// TIA Portal V20 export
FUNCTION "PMC_Map01" : Void   // FC5001, LAD
TITLE = GMPT Common Logic Template Version: G3.2
AUTHOR : JRose
FAMILY : CITI
NAME : MMG3.2
VERSION : 0.0
// stored: Namespace CITI_Logic, SetENOAutomatically false
   VAR_TEMP
      Team_Leader_Call : Bool;   // Unacknowledged Assistance Call is Active
      Flash_Red_Cmd : Bool;   // 1Hz Flasher
      Solid_Red_Cmd : Bool;   // 1Hz Flasher
      Flash_Yellow_Cmd : Bool;   // 1Hz Flasher
      Solid_Yellow_Cmd : Bool;   // 1Hz Flasher
      Flash_Green_Cmd : Bool;   // 1Hz Flasher
      Solid_Green_Cmd : Bool;   // 1Hz Flasher
      Flash_Blue_Cmd : Bool;   // 1Hz Flasher
      Solid_Blue_Cmd : Bool;   // 1Hz Flasher
      Flasher : Bool;   // 1Hz Flasher
      PUNData : String[18];
      FTQ_Reject_String : String[100];   // FTQ Data String PUN
      FTQ_Reject_Int : Int;   // FTQ Reject Integer
      LastPartTypeString : String[10];   // Last Part Type String
      EmptyPalletChar : Char;
      GM_PartNumber : String[8];
      OptionalData : String[9];
      HMI_Lite : Bool;
      HMI_Pro : Bool;
      TEMP_FOR_HMI_PRO : Bool;
      TEMP_FOR_UNIFIED_HMI : Bool;
      TEMP_HMI_INTERFACE : Bool;
      UNIFIED_HMI : Bool;
      OEM_ALARM_ID_from_ProDIAG : Int;
      Temp_Clock_Byte : Byte;
      TEMP_ALARM_FAULT : Array[0..499] of Word;
      Buffer_Count_Int : Int;
   END_VAR
   VAR_TEMP   // added for the SCL form of the ladder/FBD networks
      _w1 : Bool;
      _w2 : Bool;
      _w3 : Bool;
      _w4 : Bool;
      _w5 : Bool;
      _w6 : Bool;
      _w7 : Bool;
      _w8 : Bool;
      _w9 : Bool;
      _w10 : Bool;
      _w11 : Bool;
      _w12 : Bool;
   END_VAR
BEGIN

REGION Network 1
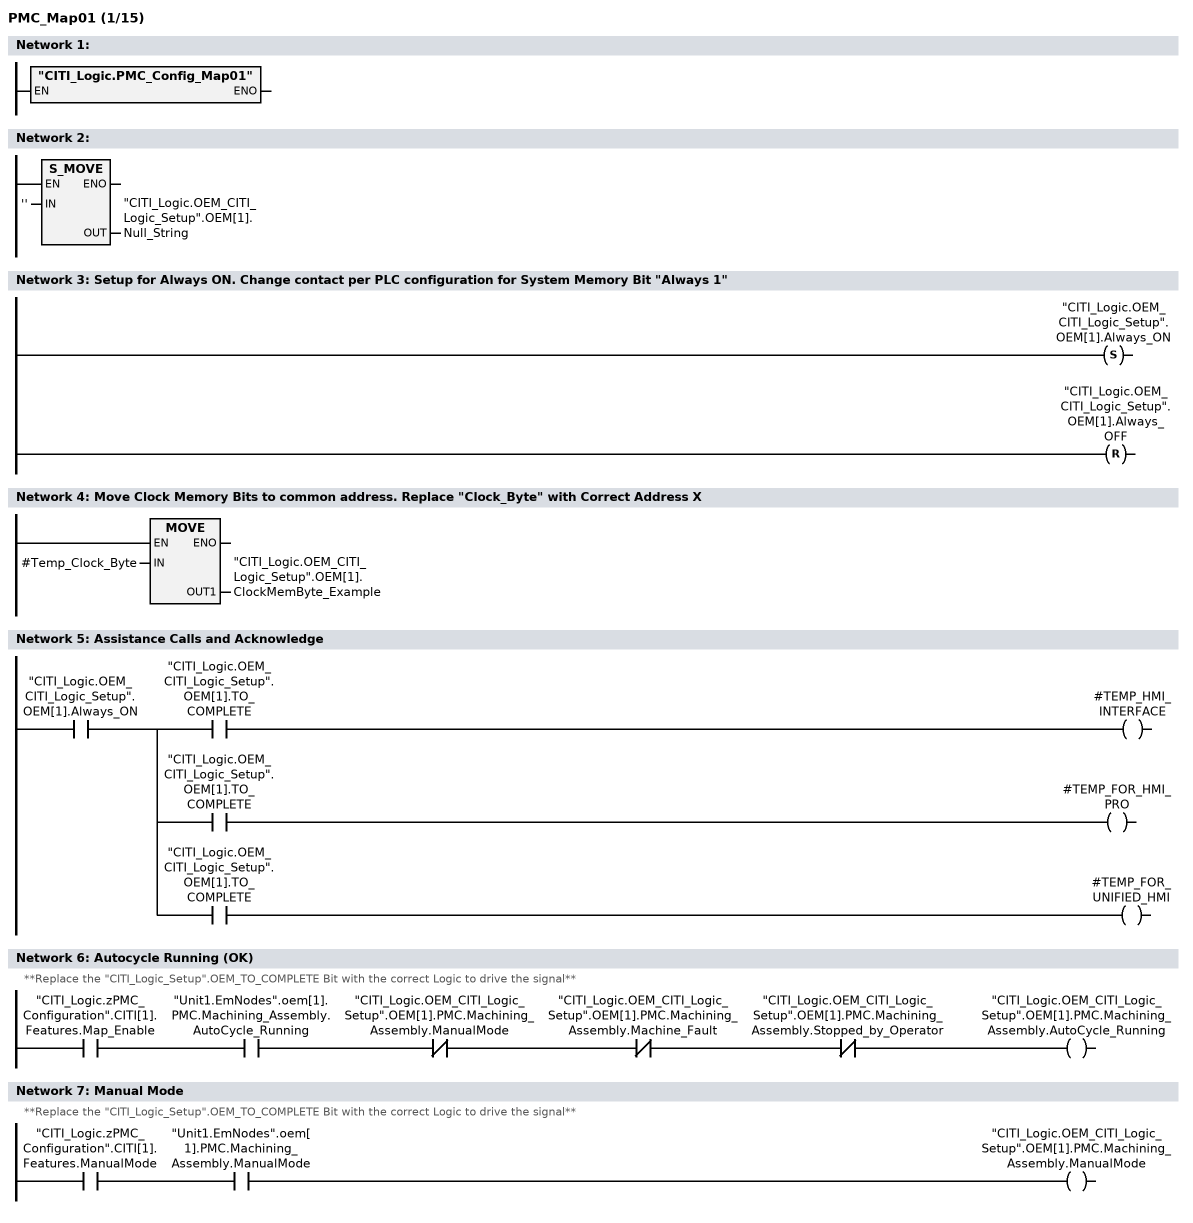
   RUNG wire#powerrail
      "CITI_Logic.PMC_Config_Map01"()
   END_RUNG
   // the same network as SCL:
   "CITI_Logic.PMC_Config_Map01"();
END_REGION

REGION Network 2
   RUNG wire#powerrail
      S_Move(in := '', out => "CITI_Logic.OEM_CITI_Logic_Setup".OEM[1].Null_String)
   END_RUNG
   // the same network as SCL:
   "CITI_Logic.OEM_CITI_Logic_Setup".OEM[1].Null_String := '';
END_REGION

REGION Network 3: Setup for Always ON. Change contact per PLC configuration for System Memory Bit "Always 1"
   RUNG wire#powerrail
      S_Coil( "CITI_Logic.OEM_CITI_Logic_Setup".OEM[1].Always_ON )
   END_RUNG
   RUNG wire#powerrail
      R_Coil( "CITI_Logic.OEM_CITI_Logic_Setup".OEM[1].Always_OFF )
   END_RUNG
   // the same network as SCL:
   "CITI_Logic.OEM_CITI_Logic_Setup".OEM[1].Always_ON := TRUE;
   "CITI_Logic.OEM_CITI_Logic_Setup".OEM[1].Always_OFF := FALSE;
END_REGION

REGION Network 4: Move Clock Memory Bits to common address. Replace "Clock_Byte" with Correct Address X
   RUNG wire#powerrail
      Move(in := #Temp_Clock_Byte, out1 => "CITI_Logic.OEM_CITI_Logic_Setup".OEM[1].ClockMemByte_Example)
   END_RUNG
   // the same network as SCL:
   "CITI_Logic.OEM_CITI_Logic_Setup".OEM[1].ClockMemByte_Example := #Temp_Clock_Byte;
END_REGION

REGION Network 5: Assistance Calls and Acknowledge
   RUNG wire#powerrail
      Contact( "CITI_Logic.OEM_CITI_Logic_Setup".OEM[1].Always_ON )
      wire#w1
      Contact( "CITI_Logic.OEM_CITI_Logic_Setup".OEM[1].TO_COMPLETE )
      Coil( #TEMP_HMI_INTERFACE )
   END_RUNG
   RUNG wire#w1
      Contact( "CITI_Logic.OEM_CITI_Logic_Setup".OEM[1].TO_COMPLETE )
      Coil( #TEMP_FOR_HMI_PRO )
   END_RUNG
   RUNG wire#w1
      Contact( "CITI_Logic.OEM_CITI_Logic_Setup".OEM[1].TO_COMPLETE )
      Coil( #TEMP_FOR_UNIFIED_HMI )
   END_RUNG
   // the same network as SCL:
   #TEMP_HMI_INTERFACE := "CITI_Logic.OEM_CITI_Logic_Setup".OEM[1].Always_ON AND "CITI_Logic.OEM_CITI_Logic_Setup".OEM[1].TO_COMPLETE;
   #TEMP_FOR_HMI_PRO := "CITI_Logic.OEM_CITI_Logic_Setup".OEM[1].Always_ON AND "CITI_Logic.OEM_CITI_Logic_Setup".OEM[1].TO_COMPLETE;
   #TEMP_FOR_UNIFIED_HMI := "CITI_Logic.OEM_CITI_Logic_Setup".OEM[1].Always_ON AND "CITI_Logic.OEM_CITI_Logic_Setup".OEM[1].TO_COMPLETE;
END_REGION

REGION Network 6: Autocycle Running (OK)
   // **Replace the "CITI_Logic_Setup".OEM_TO_COMPLETE Bit with the correct Logic to drive the signal**
   RUNG wire#powerrail
      Contact( "CITI_Logic.zPMC_Configuration".CITI[1].Features.Map_Enable )
      Contact( "Unit1.EmNodes".oem[1].PMC.Machining_Assembly.AutoCycle_Running )
      I_Contact( "CITI_Logic.OEM_CITI_Logic_Setup".OEM[1].PMC.Machining_Assembly.ManualMode )
      I_Contact( "CITI_Logic.OEM_CITI_Logic_Setup".OEM[1].PMC.Machining_Assembly.Machine_Fault )
      I_Contact( "CITI_Logic.OEM_CITI_Logic_Setup".OEM[1].PMC.Machining_Assembly.Stopped_by_Operator )
      Coil( "CITI_Logic.OEM_CITI_Logic_Setup".OEM[1].PMC.Machining_Assembly.AutoCycle_Running )
   END_RUNG
   // the same network as SCL:
   "CITI_Logic.OEM_CITI_Logic_Setup".OEM[1].PMC.Machining_Assembly.AutoCycle_Running := "CITI_Logic.zPMC_Configuration".CITI[1].Features.Map_Enable AND "Unit1.EmNodes".oem[1].PMC.Machining_Assembly.AutoCycle_Running AND NOT "CITI_Logic.OEM_CITI_Logic_Setup".OEM[1].PMC.Machining_Assembly.ManualMode AND NOT "CITI_Logic.OEM_CITI_Logic_Setup".OEM[1].PMC.Machining_Assembly.Machine_Fault AND NOT "CITI_Logic.OEM_CITI_Logic_Setup".OEM[1].PMC.Machining_Assembly.Stopped_by_Operator;
END_REGION

REGION Network 7: Manual Mode
   // **Replace the "CITI_Logic_Setup".OEM_TO_COMPLETE Bit with the correct Logic to drive the signal**
   RUNG wire#powerrail
      Contact( "CITI_Logic.zPMC_Configuration".CITI[1].Features.ManualMode )
      Contact( "Unit1.EmNodes".oem[1].PMC.Machining_Assembly.ManualMode )
      Coil( "CITI_Logic.OEM_CITI_Logic_Setup".OEM[1].PMC.Machining_Assembly.ManualMode )
   END_RUNG
   // the same network as SCL:
   "CITI_Logic.OEM_CITI_Logic_Setup".OEM[1].PMC.Machining_Assembly.ManualMode := "CITI_Logic.zPMC_Configuration".CITI[1].Features.ManualMode AND "Unit1.EmNodes".oem[1].PMC.Machining_Assembly.ManualMode;
END_REGION

REGION Network 8: Material Low (N/A)
   // **Replace the "CITI_Logic_Setup".OEM_TO_COMPLETE Bit with the correct Logic to drive the signal**
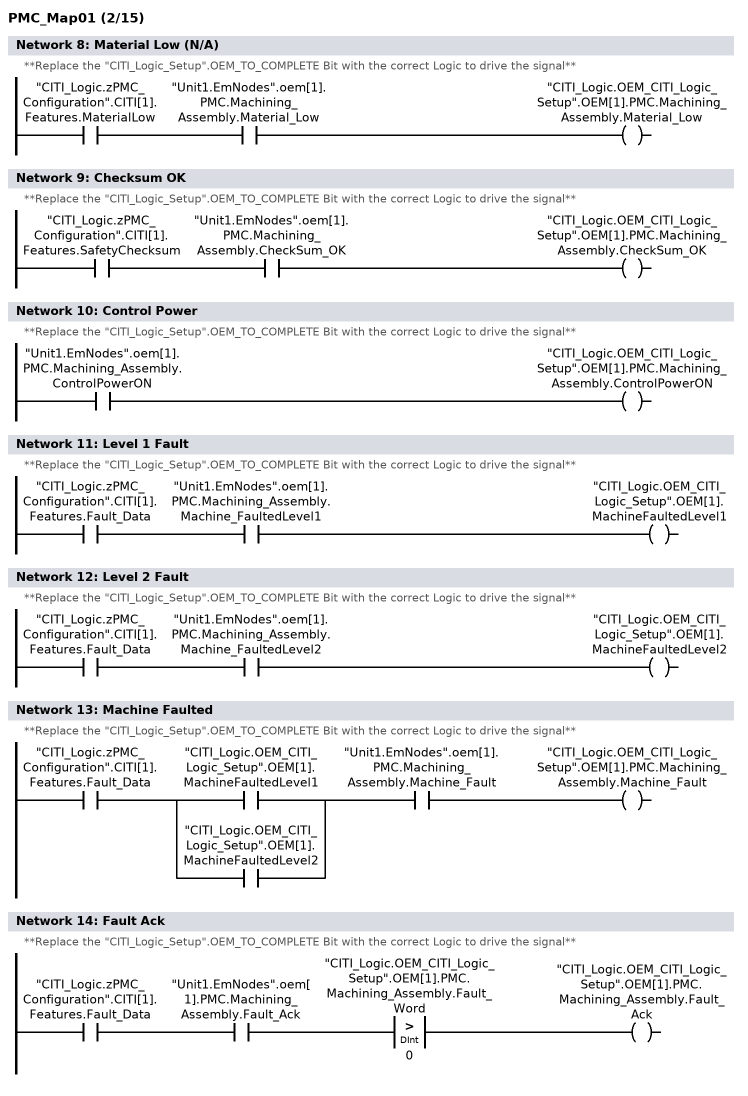
   RUNG wire#powerrail
      Contact( "CITI_Logic.zPMC_Configuration".CITI[1].Features.MaterialLow )
      Contact( "Unit1.EmNodes".oem[1].PMC.Machining_Assembly.Material_Low )
      Coil( "CITI_Logic.OEM_CITI_Logic_Setup".OEM[1].PMC.Machining_Assembly.Material_Low )
   END_RUNG
   // the same network as SCL:
   "CITI_Logic.OEM_CITI_Logic_Setup".OEM[1].PMC.Machining_Assembly.Material_Low := "CITI_Logic.zPMC_Configuration".CITI[1].Features.MaterialLow AND "Unit1.EmNodes".oem[1].PMC.Machining_Assembly.Material_Low;
END_REGION

REGION Network 9: Checksum OK
   // **Replace the "CITI_Logic_Setup".OEM_TO_COMPLETE Bit with the correct Logic to drive the signal**
   RUNG wire#powerrail
      Contact( "CITI_Logic.zPMC_Configuration".CITI[1].Features.SafetyChecksum )
      Contact( "Unit1.EmNodes".oem[1].PMC.Machining_Assembly.CheckSum_OK )
      Coil( "CITI_Logic.OEM_CITI_Logic_Setup".OEM[1].PMC.Machining_Assembly.CheckSum_OK )
   END_RUNG
   // the same network as SCL:
   "CITI_Logic.OEM_CITI_Logic_Setup".OEM[1].PMC.Machining_Assembly.CheckSum_OK := "CITI_Logic.zPMC_Configuration".CITI[1].Features.SafetyChecksum AND "Unit1.EmNodes".oem[1].PMC.Machining_Assembly.CheckSum_OK;
END_REGION

REGION Network 10: Control Power
   // **Replace the "CITI_Logic_Setup".OEM_TO_COMPLETE Bit with the correct Logic to drive the signal**
   RUNG wire#powerrail
      Contact( "Unit1.EmNodes".oem[1].PMC.Machining_Assembly.ControlPowerON )
      Coil( "CITI_Logic.OEM_CITI_Logic_Setup".OEM[1].PMC.Machining_Assembly.ControlPowerON )
   END_RUNG
   // the same network as SCL:
   "CITI_Logic.OEM_CITI_Logic_Setup".OEM[1].PMC.Machining_Assembly.ControlPowerON := "Unit1.EmNodes".oem[1].PMC.Machining_Assembly.ControlPowerON;
END_REGION

REGION Network 11: Level 1 Fault
   // **Replace the "CITI_Logic_Setup".OEM_TO_COMPLETE Bit with the correct Logic to drive the signal**
   RUNG wire#powerrail
      Contact( "CITI_Logic.zPMC_Configuration".CITI[1].Features.Fault_Data )
      Contact( "Unit1.EmNodes".oem[1].PMC.Machining_Assembly.Machine_FaultedLevel1 )
      Coil( "CITI_Logic.OEM_CITI_Logic_Setup".OEM[1].MachineFaultedLevel1 )
   END_RUNG
   // the same network as SCL:
   "CITI_Logic.OEM_CITI_Logic_Setup".OEM[1].MachineFaultedLevel1 := "CITI_Logic.zPMC_Configuration".CITI[1].Features.Fault_Data AND "Unit1.EmNodes".oem[1].PMC.Machining_Assembly.Machine_FaultedLevel1;
END_REGION

REGION Network 12: Level 2 Fault
   // **Replace the "CITI_Logic_Setup".OEM_TO_COMPLETE Bit with the correct Logic to drive the signal**
   RUNG wire#powerrail
      Contact( "CITI_Logic.zPMC_Configuration".CITI[1].Features.Fault_Data )
      Contact( "Unit1.EmNodes".oem[1].PMC.Machining_Assembly.Machine_FaultedLevel2 )
      Coil( "CITI_Logic.OEM_CITI_Logic_Setup".OEM[1].MachineFaultedLevel2 )
   END_RUNG
   // the same network as SCL:
   "CITI_Logic.OEM_CITI_Logic_Setup".OEM[1].MachineFaultedLevel2 := "CITI_Logic.zPMC_Configuration".CITI[1].Features.Fault_Data AND "Unit1.EmNodes".oem[1].PMC.Machining_Assembly.Machine_FaultedLevel2;
END_REGION

REGION Network 13: Machine Faulted
   // **Replace the "CITI_Logic_Setup".OEM_TO_COMPLETE Bit with the correct Logic to drive the signal**
   RUNG wire#powerrail
      Contact( "CITI_Logic.zPMC_Configuration".CITI[1].Features.Fault_Data )
      wire#w1
      Contact( "CITI_Logic.OEM_CITI_Logic_Setup".OEM[1].MachineFaultedLevel1 )
      wire#w2
      Contact( "Unit1.EmNodes".oem[1].PMC.Machining_Assembly.Machine_Fault )
      Coil( "CITI_Logic.OEM_CITI_Logic_Setup".OEM[1].PMC.Machining_Assembly.Machine_Fault )
   END_RUNG
   RUNG wire#w1
      Contact( "CITI_Logic.OEM_CITI_Logic_Setup".OEM[1].MachineFaultedLevel2 )
   END_RUNG wire#w2
   // the same network as SCL:
   "CITI_Logic.OEM_CITI_Logic_Setup".OEM[1].PMC.Machining_Assembly.Machine_Fault := "CITI_Logic.zPMC_Configuration".CITI[1].Features.Fault_Data AND ("CITI_Logic.OEM_CITI_Logic_Setup".OEM[1].MachineFaultedLevel1 OR "CITI_Logic.OEM_CITI_Logic_Setup".OEM[1].MachineFaultedLevel2) AND "Unit1.EmNodes".oem[1].PMC.Machining_Assembly.Machine_Fault;
END_REGION

REGION Network 14: Fault Ack
   // **Replace the "CITI_Logic_Setup".OEM_TO_COMPLETE Bit with the correct Logic to drive the signal**
   RUNG wire#powerrail
      Contact( "CITI_Logic.zPMC_Configuration".CITI[1].Features.Fault_Data )
      Contact( "Unit1.EmNodes".oem[1].PMC.Machining_Assembly.Fault_Ack )
      { S7_Templates := "SrcType := DInt" } GT_Contact(in1 := "CITI_Logic.OEM_CITI_Logic_Setup".OEM[1].PMC.Machining_Assembly.Fault_Word, in2 := 0)
      Coil( "CITI_Logic.OEM_CITI_Logic_Setup".OEM[1].PMC.Machining_Assembly.Fault_Ack )
   END_RUNG
   // the same network as SCL:
   "CITI_Logic.OEM_CITI_Logic_Setup".OEM[1].PMC.Machining_Assembly.Fault_Ack := "CITI_Logic.zPMC_Configuration".CITI[1].Features.Fault_Data AND "Unit1.EmNodes".oem[1].PMC.Machining_Assembly.Fault_Ack AND ("CITI_Logic.OEM_CITI_Logic_Setup".OEM[1].PMC.Machining_Assembly.Fault_Word > 0);
END_REGION

REGION Network 15: Stopped By Operator
   // **Replace the "CITI_Logic_Setup".OEM_TO_COMPLETE Bit with the correct Logic to drive the signal**
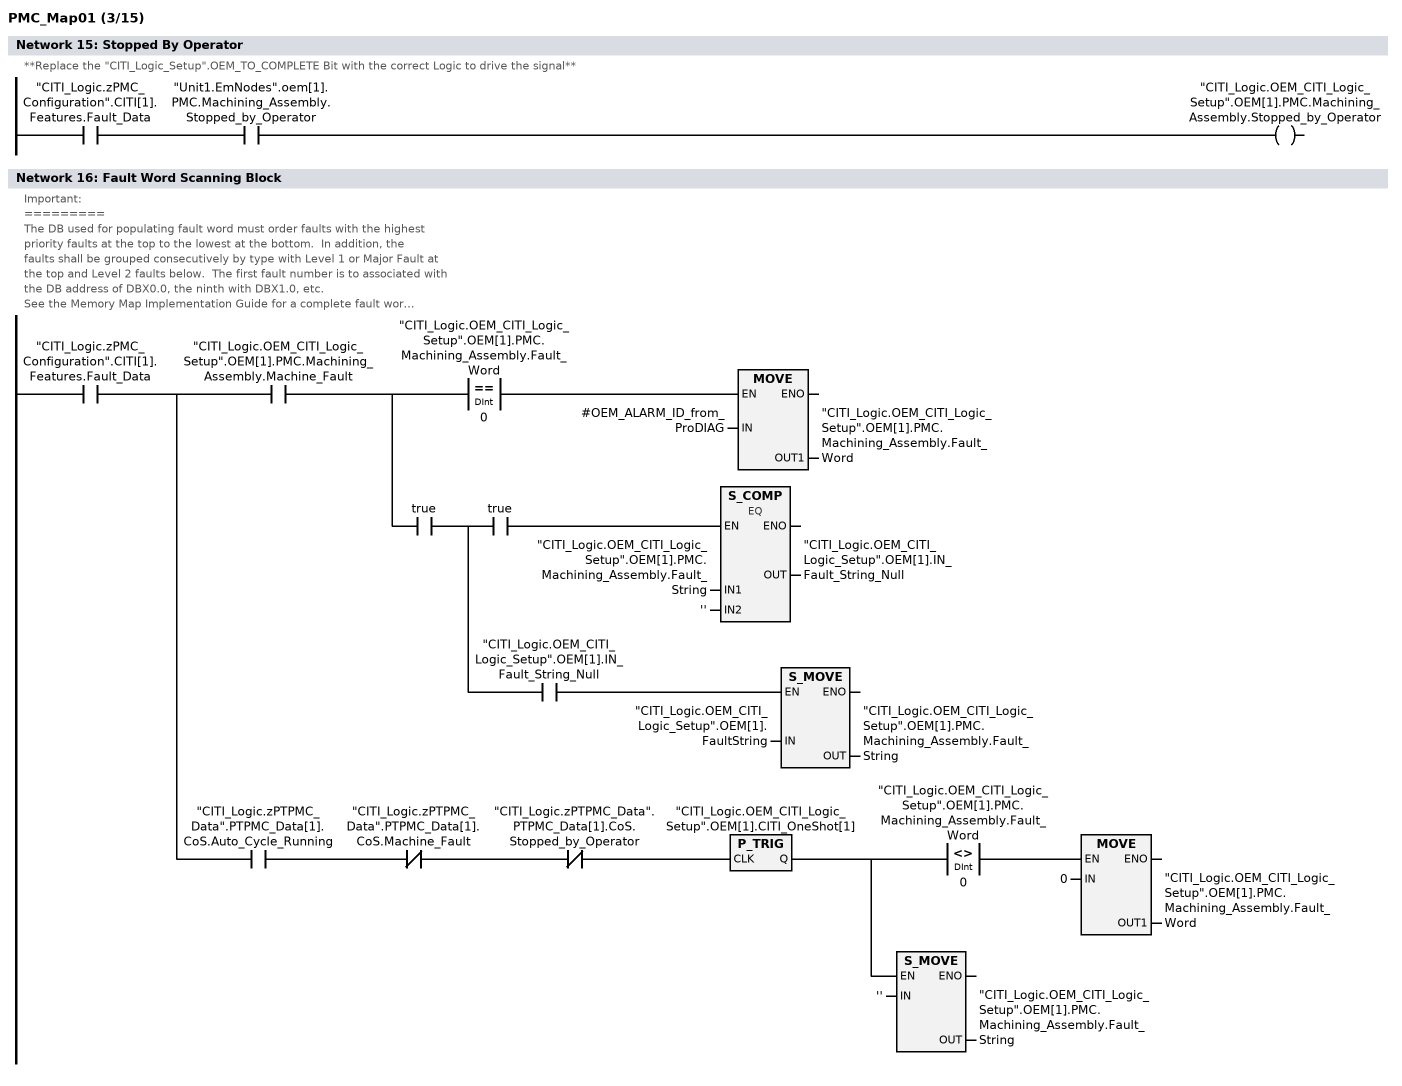
   RUNG wire#powerrail
      Contact( "CITI_Logic.zPMC_Configuration".CITI[1].Features.Fault_Data )
      Contact( "Unit1.EmNodes".oem[1].PMC.Machining_Assembly.Stopped_by_Operator )
      Coil( "CITI_Logic.OEM_CITI_Logic_Setup".OEM[1].PMC.Machining_Assembly.Stopped_by_Operator )
   END_RUNG
   // the same network as SCL:
   "CITI_Logic.OEM_CITI_Logic_Setup".OEM[1].PMC.Machining_Assembly.Stopped_by_Operator := "CITI_Logic.zPMC_Configuration".CITI[1].Features.Fault_Data AND "Unit1.EmNodes".oem[1].PMC.Machining_Assembly.Stopped_by_Operator;
END_REGION

REGION Network 16: Fault Word Scanning Block
   // Important:
   // =========
   // The DB used for populating fault word must order faults with the highest 
   // priority faults at the top to the lowest at the bottom.  In addition, the 
   // faults shall be grouped consecutively by type with Level 1 or Major Fault at 
   // the top and Level 2 faults below.  The first fault number is to associated with 
   // the DB address of DBX0.0, the ninth with DBX1.0, etc.
   // 
   // See the Memory Map Implementation Guide for a complete fault word 
   // implementation description and list of requirements.
   RUNG wire#powerrail
      Contact( "CITI_Logic.zPMC_Configuration".CITI[1].Features.Fault_Data )
      wire#w1
      Contact( "CITI_Logic.OEM_CITI_Logic_Setup".OEM[1].PMC.Machining_Assembly.Machine_Fault )
      wire#w2
      { S7_Templates := "SrcType := DInt" } EQ_Contact(in1 := "CITI_Logic.OEM_CITI_Logic_Setup".OEM[1].PMC.Machining_Assembly.Fault_Word, in2 := 0)
      Move(in := #OEM_ALARM_ID_from_ProDIAG, out1 => "CITI_Logic.OEM_CITI_Logic_Setup".OEM[1].PMC.Machining_Assembly.Fault_Word)
   END_RUNG
   RUNG wire#w2
      Contact( true )
      wire#w3
      Contact( true )
      { S7_Templates := "[relation := EQ, src_type := String]" } S_COMP(IN1 := "CITI_Logic.OEM_CITI_Logic_Setup".OEM[1].PMC.Machining_Assembly.Fault_String, IN2 := '', OUT => "CITI_Logic.OEM_CITI_Logic_Setup".OEM[1].IN_Fault_String_Null)
   END_RUNG
   RUNG wire#w3
      Contact( "CITI_Logic.OEM_CITI_Logic_Setup".OEM[1].IN_Fault_String_Null )
      S_Move(in := "CITI_Logic.OEM_CITI_Logic_Setup".OEM[1].FaultString, out => "CITI_Logic.OEM_CITI_Logic_Setup".OEM[1].PMC.Machining_Assembly.Fault_String)
   END_RUNG
   RUNG wire#w1
      Contact( "CITI_Logic.zPTPMC_Data".PTPMC_Data[1].CoS.Auto_Cycle_Running )
      I_Contact( "CITI_Logic.zPTPMC_Data".PTPMC_Data[1].CoS.Machine_Fault )
      I_Contact( "CITI_Logic.zPTPMC_Data".PTPMC_Data[1].CoS.Stopped_by_Operator )
      P_Trig( "CITI_Logic.OEM_CITI_Logic_Setup".OEM[1].CITI_OneShot[1] )
      wire#w4
      { S7_Templates := "SrcType := DInt" } NE_Contact(in1 := "CITI_Logic.OEM_CITI_Logic_Setup".OEM[1].PMC.Machining_Assembly.Fault_Word, in2 := 0)
      { S7_GenerateENO := "TRUE" } Move(in := 0, out1 => "CITI_Logic.OEM_CITI_Logic_Setup".OEM[1].PMC.Machining_Assembly.Fault_Word)
   END_RUNG
   RUNG wire#w4
      S_Move(in := '', out => "CITI_Logic.OEM_CITI_Logic_Setup".OEM[1].PMC.Machining_Assembly.Fault_String)
   END_RUNG
   // the same network as SCL:
   #_w1 := "CITI_Logic.zPMC_Configuration".CITI[1].Features.Fault_Data AND "CITI_Logic.OEM_CITI_Logic_Setup".OEM[1].PMC.Machining_Assembly.Machine_Fault;
   IF #_w1 AND ("CITI_Logic.OEM_CITI_Logic_Setup".OEM[1].PMC.Machining_Assembly.Fault_Word = 0) THEN
       "CITI_Logic.OEM_CITI_Logic_Setup".OEM[1].PMC.Machining_Assembly.Fault_Word := #OEM_ALARM_ID_from_ProDIAG;
   END_IF;
   #_w2 := #_w1 AND true;
   #_w3 := "CITI_Logic.zPMC_Configuration".CITI[1].Features.Fault_Data;
   IF #_w2 AND true THEN
       S_COMP(IN1 := "CITI_Logic.OEM_CITI_Logic_Setup".OEM[1].PMC.Machining_Assembly.Fault_String,
              IN2 := '',
              OUT => "CITI_Logic.OEM_CITI_Logic_Setup".OEM[1].IN_Fault_String_Null);
   END_IF;
   IF #_w2 AND "CITI_Logic.OEM_CITI_Logic_Setup".OEM[1].IN_Fault_String_Null THEN
       "CITI_Logic.OEM_CITI_Logic_Setup".OEM[1].PMC.Machining_Assembly.Fault_String := "CITI_Logic.OEM_CITI_Logic_Setup".OEM[1].FaultString;
   END_IF;
   #_w4 := #_w3 AND "CITI_Logic.zPTPMC_Data".PTPMC_Data[1].CoS.Auto_Cycle_Running AND NOT "CITI_Logic.zPTPMC_Data".PTPMC_Data[1].CoS.Machine_Fault AND NOT "CITI_Logic.zPTPMC_Data".PTPMC_Data[1].CoS.Stopped_by_Operator;
   #_w5 := #_w4 AND NOT "CITI_Logic.OEM_CITI_Logic_Setup".OEM[1].CITI_OneShot[1];   // rising edge
   "CITI_Logic.OEM_CITI_Logic_Setup".OEM[1].CITI_OneShot[1] := #_w4;
   IF #_w5 AND ("CITI_Logic.OEM_CITI_Logic_Setup".OEM[1].PMC.Machining_Assembly.Fault_Word <> 0) THEN
       "CITI_Logic.OEM_CITI_Logic_Setup".OEM[1].PMC.Machining_Assembly.Fault_Word := 0;
   END_IF;
   IF #_w5 THEN "CITI_Logic.OEM_CITI_Logic_Setup".OEM[1].PMC.Machining_Assembly.Fault_String := ''; END_IF;
END_REGION

REGION Network 17: Set up for Stopped by Other Map or Stopped with Unknown Fault
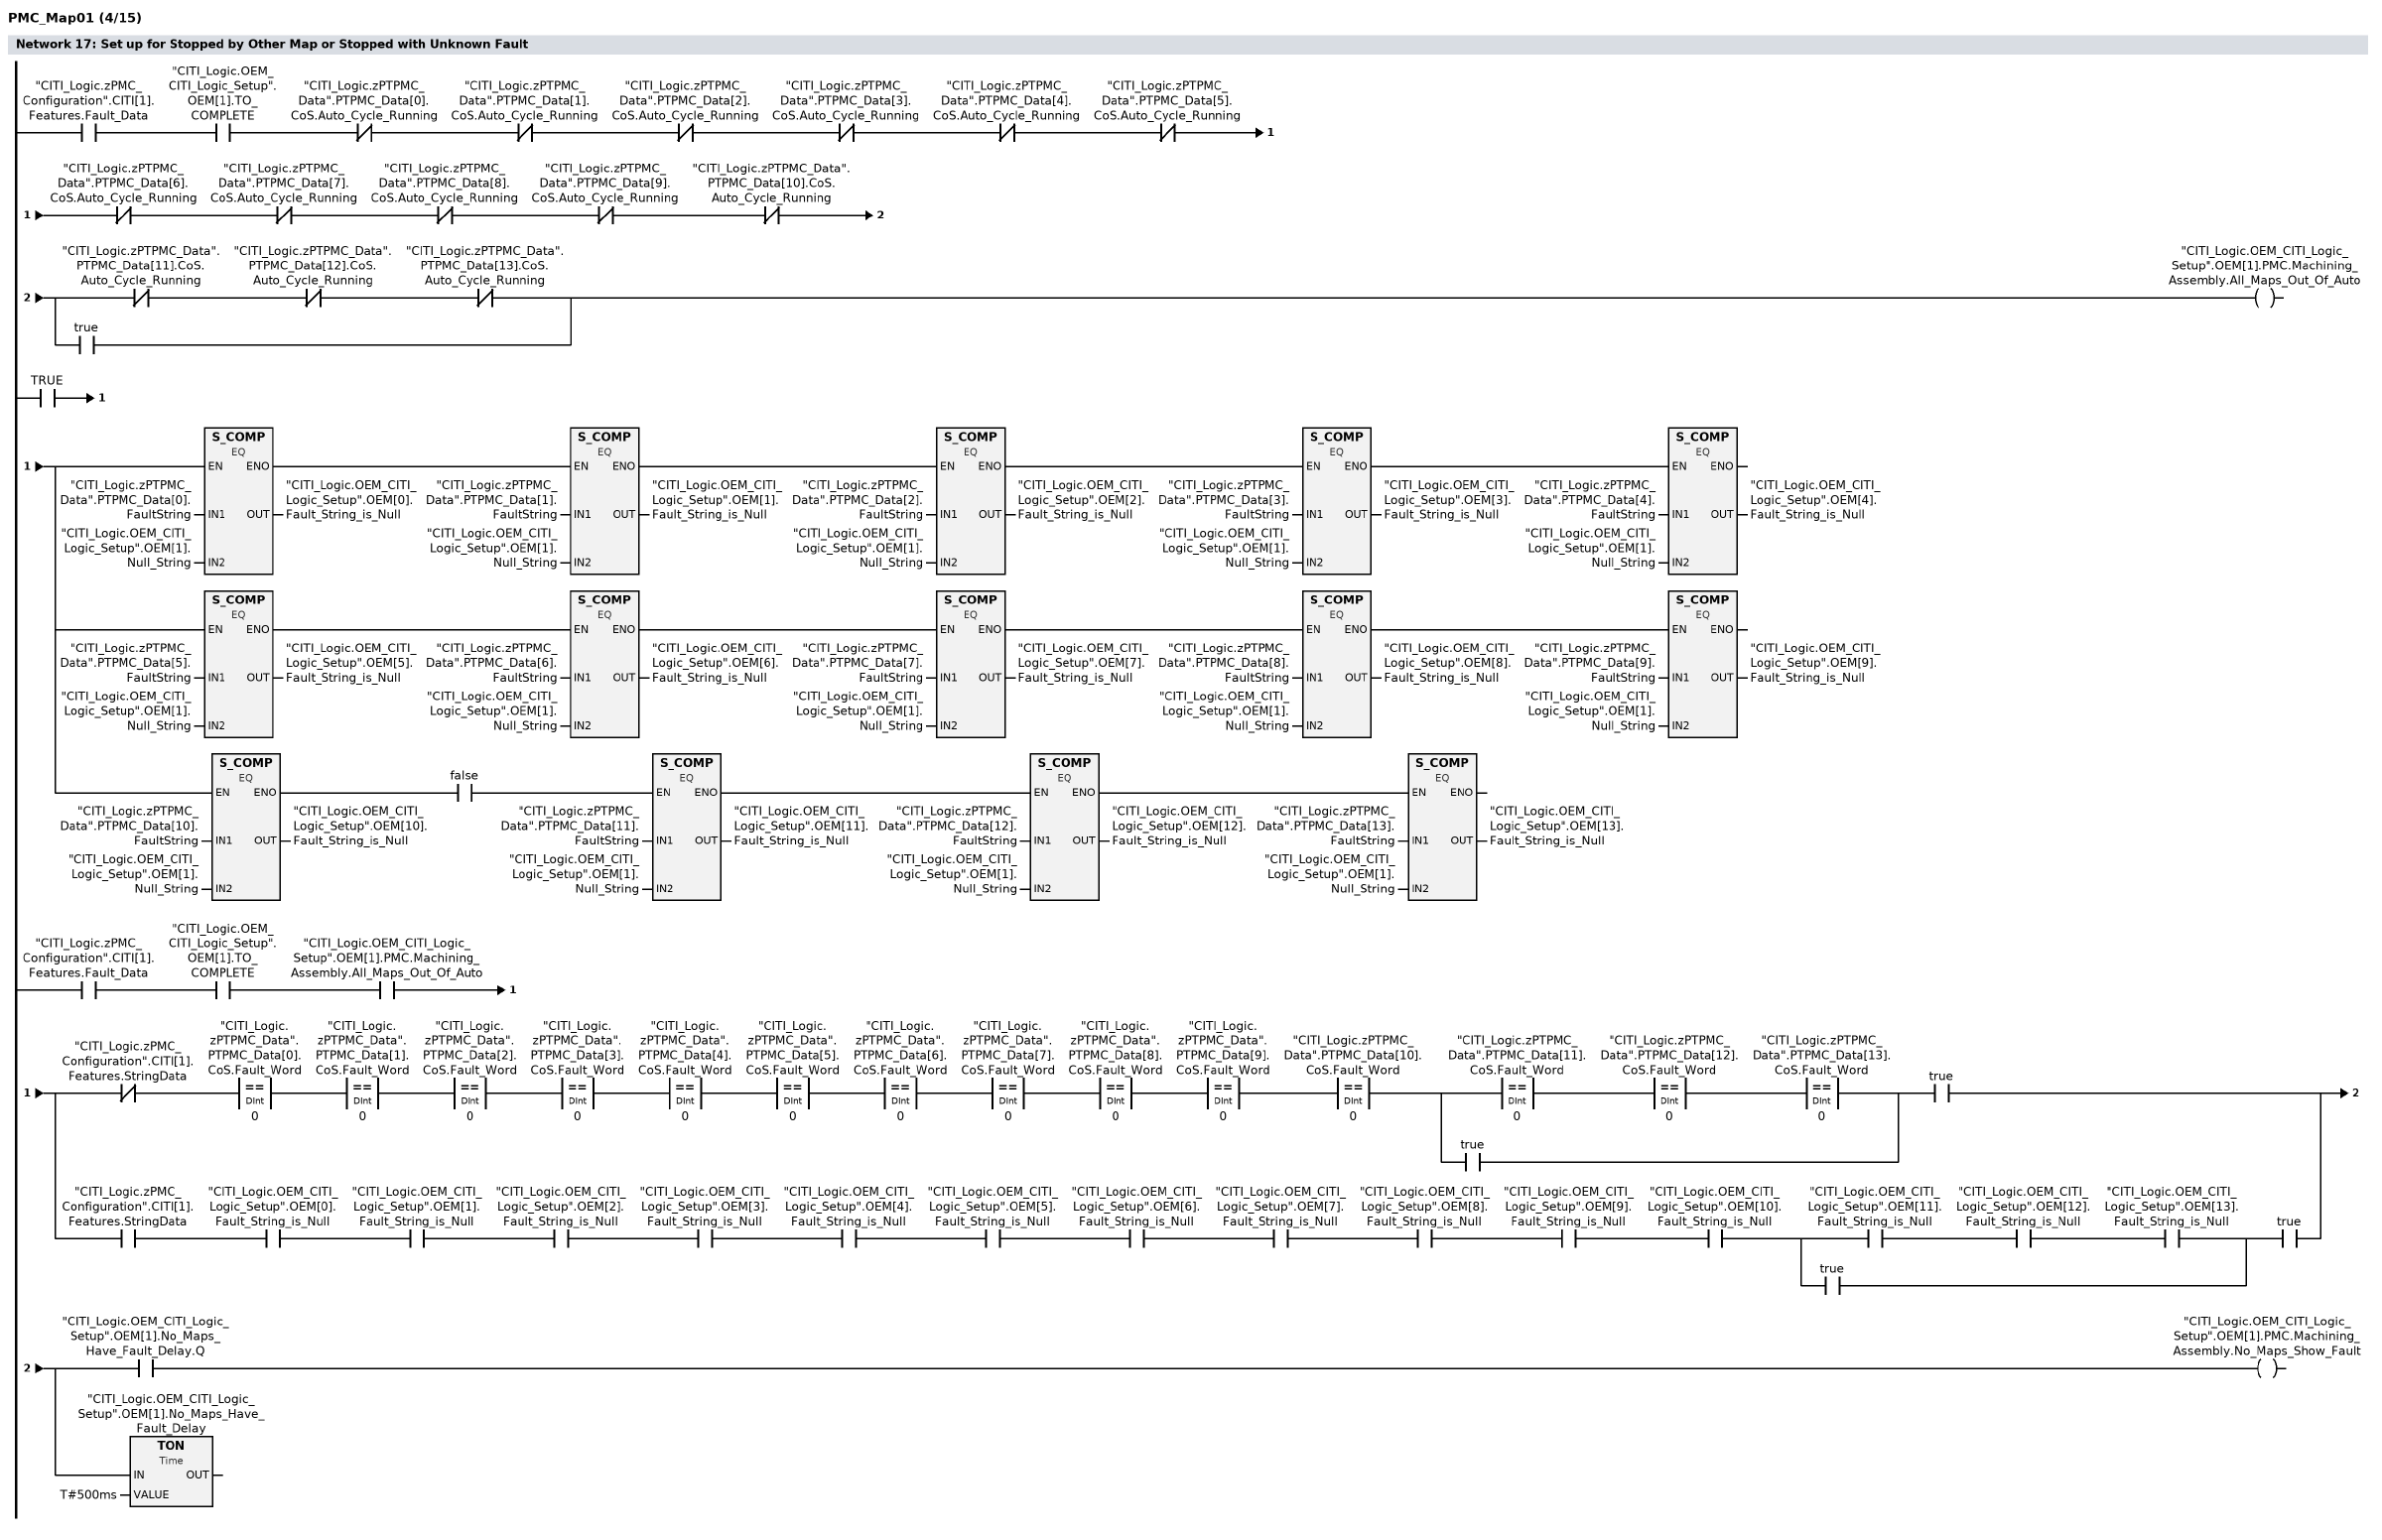
   "CITI_Logic.OEM_CITI_Logic_Setup".OEM[1].PMC.Machining_Assembly.All_Maps_Out_Of_Auto := "CITI_Logic.zPMC_Configuration".CITI[1].Features.Fault_Data AND "CITI_Logic.OEM_CITI_Logic_Setup".OEM[1].TO_COMPLETE AND NOT "CITI_Logic.zPTPMC_Data".PTPMC_Data[0].CoS.Auto_Cycle_Running AND NOT "CITI_Logic.zPTPMC_Data".PTPMC_Data[1].CoS.Auto_Cycle_Running AND NOT "CITI_Logic.zPTPMC_Data".PTPMC_Data[2].CoS.Auto_Cycle_Running AND NOT "CITI_Logic.zPTPMC_Data".PTPMC_Data[3].CoS.Auto_Cycle_Running AND NOT "CITI_Logic.zPTPMC_Data".PTPMC_Data[4].CoS.Auto_Cycle_Running AND NOT "CITI_Logic.zPTPMC_Data".PTPMC_Data[5].CoS.Auto_Cycle_Running AND NOT "CITI_Logic.zPTPMC_Data".PTPMC_Data[6].CoS.Auto_Cycle_Running AND NOT "CITI_Logic.zPTPMC_Data".PTPMC_Data[7].CoS.Auto_Cycle_Running AND NOT "CITI_Logic.zPTPMC_Data".PTPMC_Data[8].CoS.Auto_Cycle_Running AND NOT "CITI_Logic.zPTPMC_Data".PTPMC_Data[9].CoS.Auto_Cycle_Running AND NOT "CITI_Logic.zPTPMC_Data".PTPMC_Data[10].CoS.Auto_Cycle_Running AND ((NOT "CITI_Logic.zPTPMC_Data".PTPMC_Data[11].CoS.Auto_Cycle_Running AND NOT "CITI_Logic.zPTPMC_Data".PTPMC_Data[12].CoS.Auto_Cycle_Running AND NOT "CITI_Logic.zPTPMC_Data".PTPMC_Data[13].CoS.Auto_Cycle_Running) OR true);
   S_COMP(EN := TRUE,
          IN1 := "CITI_Logic.zPTPMC_Data".PTPMC_Data[0].FaultString,
          IN2 := "CITI_Logic.OEM_CITI_Logic_Setup".OEM[1].Null_String,
          OUT => "CITI_Logic.OEM_CITI_Logic_Setup".OEM[0].Fault_String_is_Null,
          ENO => #_w1);
   S_COMP(EN := #_w1,
          IN1 := "CITI_Logic.zPTPMC_Data".PTPMC_Data[1].FaultString,
          IN2 := "CITI_Logic.OEM_CITI_Logic_Setup".OEM[1].Null_String,
          OUT => "CITI_Logic.OEM_CITI_Logic_Setup".OEM[1].Fault_String_is_Null,
          ENO => #_w2);
   S_COMP(EN := #_w2,
          IN1 := "CITI_Logic.zPTPMC_Data".PTPMC_Data[2].FaultString,
          IN2 := "CITI_Logic.OEM_CITI_Logic_Setup".OEM[1].Null_String,
          OUT => "CITI_Logic.OEM_CITI_Logic_Setup".OEM[2].Fault_String_is_Null,
          ENO => #_w3);
   S_COMP(EN := #_w3,
          IN1 := "CITI_Logic.zPTPMC_Data".PTPMC_Data[3].FaultString,
          IN2 := "CITI_Logic.OEM_CITI_Logic_Setup".OEM[1].Null_String,
          OUT => "CITI_Logic.OEM_CITI_Logic_Setup".OEM[3].Fault_String_is_Null,
          ENO => #_w4);
   IF #_w4 THEN
       S_COMP(IN1 := "CITI_Logic.zPTPMC_Data".PTPMC_Data[4].FaultString,
              IN2 := "CITI_Logic.OEM_CITI_Logic_Setup".OEM[1].Null_String,
              OUT => "CITI_Logic.OEM_CITI_Logic_Setup".OEM[4].Fault_String_is_Null);
   END_IF;
   S_COMP(EN := TRUE,
          IN1 := "CITI_Logic.zPTPMC_Data".PTPMC_Data[5].FaultString,
          IN2 := "CITI_Logic.OEM_CITI_Logic_Setup".OEM[1].Null_String,
          OUT => "CITI_Logic.OEM_CITI_Logic_Setup".OEM[5].Fault_String_is_Null,
          ENO => #_w5);
   S_COMP(EN := #_w5,
          IN1 := "CITI_Logic.zPTPMC_Data".PTPMC_Data[6].FaultString,
          IN2 := "CITI_Logic.OEM_CITI_Logic_Setup".OEM[1].Null_String,
          OUT => "CITI_Logic.OEM_CITI_Logic_Setup".OEM[6].Fault_String_is_Null,
          ENO => #_w6);
   S_COMP(EN := #_w6,
          IN1 := "CITI_Logic.zPTPMC_Data".PTPMC_Data[7].FaultString,
          IN2 := "CITI_Logic.OEM_CITI_Logic_Setup".OEM[1].Null_String,
          OUT => "CITI_Logic.OEM_CITI_Logic_Setup".OEM[7].Fault_String_is_Null,
          ENO => #_w7);
   S_COMP(EN := #_w7,
          IN1 := "CITI_Logic.zPTPMC_Data".PTPMC_Data[8].FaultString,
          IN2 := "CITI_Logic.OEM_CITI_Logic_Setup".OEM[1].Null_String,
          OUT => "CITI_Logic.OEM_CITI_Logic_Setup".OEM[8].Fault_String_is_Null,
          ENO => #_w8);
   IF #_w8 THEN
       S_COMP(IN1 := "CITI_Logic.zPTPMC_Data".PTPMC_Data[9].FaultString,
              IN2 := "CITI_Logic.OEM_CITI_Logic_Setup".OEM[1].Null_String,
              OUT => "CITI_Logic.OEM_CITI_Logic_Setup".OEM[9].Fault_String_is_Null);
   END_IF;
   S_COMP(EN := TRUE,
          IN1 := "CITI_Logic.zPTPMC_Data".PTPMC_Data[10].FaultString,
          IN2 := "CITI_Logic.OEM_CITI_Logic_Setup".OEM[1].Null_String,
          OUT => "CITI_Logic.OEM_CITI_Logic_Setup".OEM[10].Fault_String_is_Null,
          ENO => #_w9);
   S_COMP(EN := #_w9 AND false,
          IN1 := "CITI_Logic.zPTPMC_Data".PTPMC_Data[11].FaultString,
          IN2 := "CITI_Logic.OEM_CITI_Logic_Setup".OEM[1].Null_String,
          OUT => "CITI_Logic.OEM_CITI_Logic_Setup".OEM[11].Fault_String_is_Null,
          ENO => #_w10);
   S_COMP(EN := #_w10,
          IN1 := "CITI_Logic.zPTPMC_Data".PTPMC_Data[12].FaultString,
          IN2 := "CITI_Logic.OEM_CITI_Logic_Setup".OEM[1].Null_String,
          OUT => "CITI_Logic.OEM_CITI_Logic_Setup".OEM[12].Fault_String_is_Null,
          ENO => #_w11);
   IF #_w11 THEN
       S_COMP(IN1 := "CITI_Logic.zPTPMC_Data".PTPMC_Data[13].FaultString,
              IN2 := "CITI_Logic.OEM_CITI_Logic_Setup".OEM[1].Null_String,
              OUT => "CITI_Logic.OEM_CITI_Logic_Setup".OEM[13].Fault_String_is_Null);
   END_IF;
   #_w12 := "CITI_Logic.zPMC_Configuration".CITI[1].Features.Fault_Data AND "CITI_Logic.OEM_CITI_Logic_Setup".OEM[1].TO_COMPLETE AND "CITI_Logic.OEM_CITI_Logic_Setup".OEM[1].PMC.Machining_Assembly.All_Maps_Out_Of_Auto AND ((NOT "CITI_Logic.zPMC_Configuration".CITI[1].Features.StringData AND ("CITI_Logic.zPTPMC_Data".PTPMC_Data[0].CoS.Fault_Word = 0) AND ("CITI_Logic.zPTPMC_Data".PTPMC_Data[1].CoS.Fault_Word = 0) AND ("CITI_Logic.zPTPMC_Data".PTPMC_Data[2].CoS.Fault_Word = 0) AND ("CITI_Logic.zPTPMC_Data".PTPMC_Data[3].CoS.Fault_Word = 0) AND ("CITI_Logic.zPTPMC_Data".PTPMC_Data[4].CoS.Fault_Word = 0) AND ("CITI_Logic.zPTPMC_Data".PTPMC_Data[5].CoS.Fault_Word = 0) AND ("CITI_Logic.zPTPMC_Data".PTPMC_Data[6].CoS.Fault_Word = 0) AND ("CITI_Logic.zPTPMC_Data".PTPMC_Data[7].CoS.Fault_Word = 0) AND ("CITI_Logic.zPTPMC_Data".PTPMC_Data[8].CoS.Fault_Word = 0) AND ("CITI_Logic.zPTPMC_Data".PTPMC_Data[9].CoS.Fault_Word = 0) AND ("CITI_Logic.zPTPMC_Data".PTPMC_Data[10].CoS.Fault_Word = 0) AND ((("CITI_Logic.zPTPMC_Data".PTPMC_Data[11].CoS.Fault_Word = 0) AND ("CITI_Logic.zPTPMC_Data".PTPMC_Data[12].CoS.Fault_Word = 0) AND ("CITI_Logic.zPTPMC_Data".PTPMC_Data[13].CoS.Fault_Word = 0)) OR true) AND true) OR ("CITI_Logic.zPMC_Configuration".CITI[1].Features.StringData AND "CITI_Logic.OEM_CITI_Logic_Setup".OEM[0].Fault_String_is_Null AND "CITI_Logic.OEM_CITI_Logic_Setup".OEM[1].Fault_String_is_Null AND "CITI_Logic.OEM_CITI_Logic_Setup".OEM[2].Fault_String_is_Null AND "CITI_Logic.OEM_CITI_Logic_Setup".OEM[3].Fault_String_is_Null AND "CITI_Logic.OEM_CITI_Logic_Setup".OEM[4].Fault_String_is_Null AND "CITI_Logic.OEM_CITI_Logic_Setup".OEM[5].Fault_String_is_Null AND "CITI_Logic.OEM_CITI_Logic_Setup".OEM[6].Fault_String_is_Null AND "CITI_Logic.OEM_CITI_Logic_Setup".OEM[7].Fault_String_is_Null AND "CITI_Logic.OEM_CITI_Logic_Setup".OEM[8].Fault_String_is_Null AND "CITI_Logic.OEM_CITI_Logic_Setup".OEM[9].Fault_String_is_Null AND "CITI_Logic.OEM_CITI_Logic_Setup".OEM[10].Fault_String_is_Null AND (("CITI_Logic.OEM_CITI_Logic_Setup".OEM[11].Fault_String_is_Null AND "CITI_Logic.OEM_CITI_Logic_Setup".OEM[12].Fault_String_is_Null AND "CITI_Logic.OEM_CITI_Logic_Setup".OEM[13].Fault_String_is_Null) OR true) AND true));
   "CITI_Logic.OEM_CITI_Logic_Setup".OEM[1].PMC.Machining_Assembly.No_Maps_Show_Fault := #_w12 AND "CITI_Logic.OEM_CITI_Logic_Setup".OEM[1].No_Maps_Have_Fault_Delay.Q;
   "CITI_Logic.OEM_CITI_Logic_Setup".OEM[1].No_Maps_Have_Fault_Delay.TON(IN := #_w12, PT := T#500ms);   // TON coil
END_REGION

REGION Network 18: Dry Cycle Mode
   // **Replace the "CITI_Logic_Setup".OEM_TO_COMPLETE Bit with the correct Logic to drive the signal**
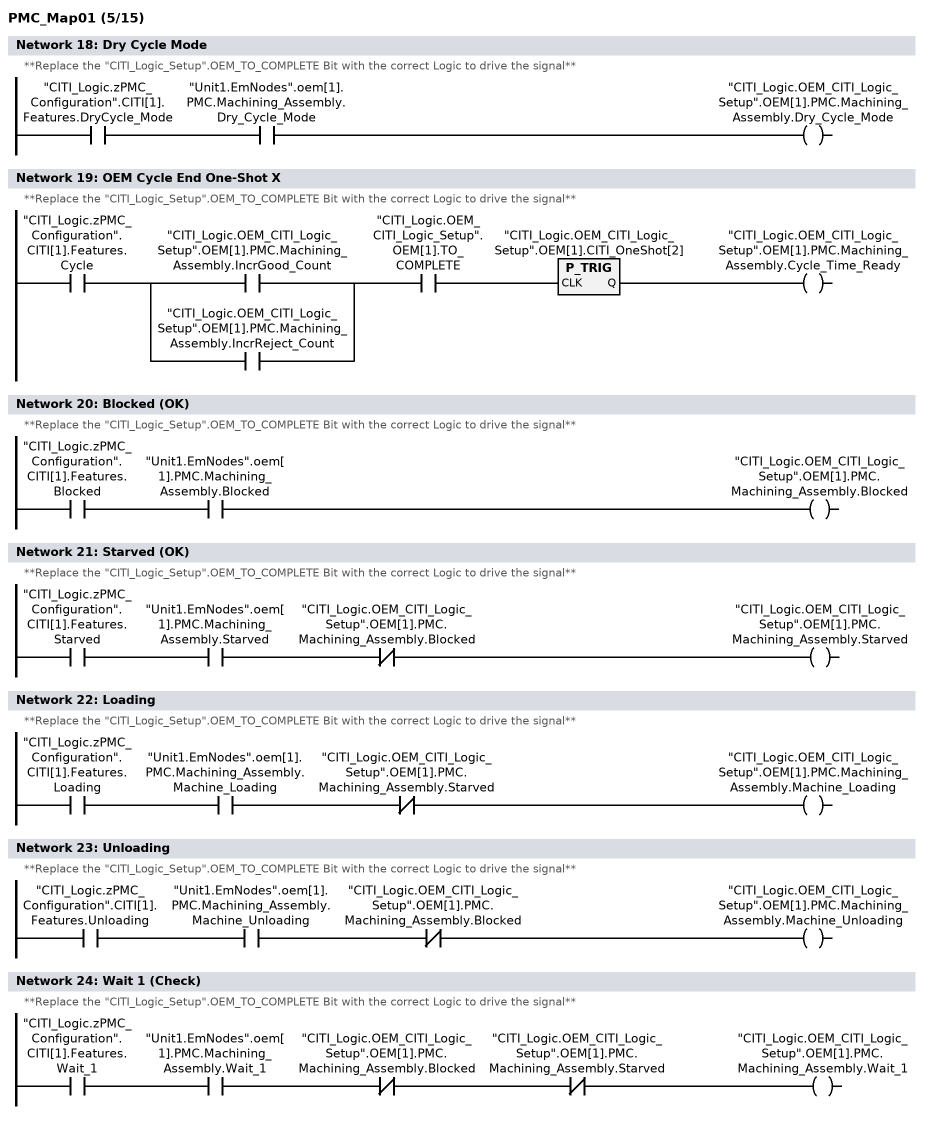
   RUNG wire#powerrail
      Contact( "CITI_Logic.zPMC_Configuration".CITI[1].Features.DryCycle_Mode )
      Contact( "Unit1.EmNodes".oem[1].PMC.Machining_Assembly.Dry_Cycle_Mode )
      Coil( "CITI_Logic.OEM_CITI_Logic_Setup".OEM[1].PMC.Machining_Assembly.Dry_Cycle_Mode )
   END_RUNG
   // the same network as SCL:
   "CITI_Logic.OEM_CITI_Logic_Setup".OEM[1].PMC.Machining_Assembly.Dry_Cycle_Mode := "CITI_Logic.zPMC_Configuration".CITI[1].Features.DryCycle_Mode AND "Unit1.EmNodes".oem[1].PMC.Machining_Assembly.Dry_Cycle_Mode;
END_REGION

REGION Network 19: OEM Cycle End One-Shot X
   // **Replace the "CITI_Logic_Setup".OEM_TO_COMPLETE Bit with the correct Logic to drive the signal**
   RUNG wire#powerrail
      Contact( "CITI_Logic.zPMC_Configuration".CITI[1].Features.Cycle )
      wire#w1
      Contact( "CITI_Logic.OEM_CITI_Logic_Setup".OEM[1].PMC.Machining_Assembly.IncrGood_Count )
      wire#w2
      Contact( "CITI_Logic.OEM_CITI_Logic_Setup".OEM[1].TO_COMPLETE )
      P_Trig( "CITI_Logic.OEM_CITI_Logic_Setup".OEM[1].CITI_OneShot[2] )
      Coil( "CITI_Logic.OEM_CITI_Logic_Setup".OEM[1].PMC.Machining_Assembly.Cycle_Time_Ready )
   END_RUNG
   RUNG wire#w1
      Contact( "CITI_Logic.OEM_CITI_Logic_Setup".OEM[1].PMC.Machining_Assembly.IncrReject_Count )
   END_RUNG wire#w2
   // the same network as SCL:
   #_w1 := "CITI_Logic.zPMC_Configuration".CITI[1].Features.Cycle AND ("CITI_Logic.OEM_CITI_Logic_Setup".OEM[1].PMC.Machining_Assembly.IncrGood_Count OR "CITI_Logic.OEM_CITI_Logic_Setup".OEM[1].PMC.Machining_Assembly.IncrReject_Count) AND "CITI_Logic.OEM_CITI_Logic_Setup".OEM[1].TO_COMPLETE;
   #_w2 := #_w1 AND NOT "CITI_Logic.OEM_CITI_Logic_Setup".OEM[1].CITI_OneShot[2];   // rising edge
   "CITI_Logic.OEM_CITI_Logic_Setup".OEM[1].CITI_OneShot[2] := #_w1;
   "CITI_Logic.OEM_CITI_Logic_Setup".OEM[1].PMC.Machining_Assembly.Cycle_Time_Ready := #_w2;
END_REGION

REGION Network 20: Blocked (OK)
   // **Replace the "CITI_Logic_Setup".OEM_TO_COMPLETE Bit with the correct Logic to drive the signal**
   RUNG wire#powerrail
      Contact( "CITI_Logic.zPMC_Configuration".CITI[1].Features.Blocked )
      Contact( "Unit1.EmNodes".oem[1].PMC.Machining_Assembly.Blocked )
      Coil( "CITI_Logic.OEM_CITI_Logic_Setup".OEM[1].PMC.Machining_Assembly.Blocked )
   END_RUNG
   // the same network as SCL:
   "CITI_Logic.OEM_CITI_Logic_Setup".OEM[1].PMC.Machining_Assembly.Blocked := "CITI_Logic.zPMC_Configuration".CITI[1].Features.Blocked AND "Unit1.EmNodes".oem[1].PMC.Machining_Assembly.Blocked;
END_REGION

REGION Network 21: Starved (OK)
   // **Replace the "CITI_Logic_Setup".OEM_TO_COMPLETE Bit with the correct Logic to drive the signal**
   RUNG wire#powerrail
      Contact( "CITI_Logic.zPMC_Configuration".CITI[1].Features.Starved )
      Contact( "Unit1.EmNodes".oem[1].PMC.Machining_Assembly.Starved )
      I_Contact( "CITI_Logic.OEM_CITI_Logic_Setup".OEM[1].PMC.Machining_Assembly.Blocked )
      Coil( "CITI_Logic.OEM_CITI_Logic_Setup".OEM[1].PMC.Machining_Assembly.Starved )
   END_RUNG
   // the same network as SCL:
   "CITI_Logic.OEM_CITI_Logic_Setup".OEM[1].PMC.Machining_Assembly.Starved := "CITI_Logic.zPMC_Configuration".CITI[1].Features.Starved AND "Unit1.EmNodes".oem[1].PMC.Machining_Assembly.Starved AND NOT "CITI_Logic.OEM_CITI_Logic_Setup".OEM[1].PMC.Machining_Assembly.Blocked;
END_REGION

REGION Network 22: Loading
   // **Replace the "CITI_Logic_Setup".OEM_TO_COMPLETE Bit with the correct Logic to drive the signal**
   RUNG wire#powerrail
      Contact( "CITI_Logic.zPMC_Configuration".CITI[1].Features.Loading )
      Contact( "Unit1.EmNodes".oem[1].PMC.Machining_Assembly.Machine_Loading )
      I_Contact( "CITI_Logic.OEM_CITI_Logic_Setup".OEM[1].PMC.Machining_Assembly.Starved )
      Coil( "CITI_Logic.OEM_CITI_Logic_Setup".OEM[1].PMC.Machining_Assembly.Machine_Loading )
   END_RUNG
   // the same network as SCL:
   "CITI_Logic.OEM_CITI_Logic_Setup".OEM[1].PMC.Machining_Assembly.Machine_Loading := "CITI_Logic.zPMC_Configuration".CITI[1].Features.Loading AND "Unit1.EmNodes".oem[1].PMC.Machining_Assembly.Machine_Loading AND NOT "CITI_Logic.OEM_CITI_Logic_Setup".OEM[1].PMC.Machining_Assembly.Starved;
END_REGION

REGION Network 23: Unloading
   // **Replace the "CITI_Logic_Setup".OEM_TO_COMPLETE Bit with the correct Logic to drive the signal**
   RUNG wire#powerrail
      Contact( "CITI_Logic.zPMC_Configuration".CITI[1].Features.Unloading )
      Contact( "Unit1.EmNodes".oem[1].PMC.Machining_Assembly.Machine_Unloading )
      I_Contact( "CITI_Logic.OEM_CITI_Logic_Setup".OEM[1].PMC.Machining_Assembly.Blocked )
      Coil( "CITI_Logic.OEM_CITI_Logic_Setup".OEM[1].PMC.Machining_Assembly.Machine_Unloading )
   END_RUNG
   // the same network as SCL:
   "CITI_Logic.OEM_CITI_Logic_Setup".OEM[1].PMC.Machining_Assembly.Machine_Unloading := "CITI_Logic.zPMC_Configuration".CITI[1].Features.Unloading AND "Unit1.EmNodes".oem[1].PMC.Machining_Assembly.Machine_Unloading AND NOT "CITI_Logic.OEM_CITI_Logic_Setup".OEM[1].PMC.Machining_Assembly.Blocked;
END_REGION

REGION Network 24: Wait 1 (Check)
   // **Replace the "CITI_Logic_Setup".OEM_TO_COMPLETE Bit with the correct Logic to drive the signal**
   RUNG wire#powerrail
      Contact( "CITI_Logic.zPMC_Configuration".CITI[1].Features.Wait_1 )
      Contact( "Unit1.EmNodes".oem[1].PMC.Machining_Assembly.Wait_1 )
      I_Contact( "CITI_Logic.OEM_CITI_Logic_Setup".OEM[1].PMC.Machining_Assembly.Blocked )
      I_Contact( "CITI_Logic.OEM_CITI_Logic_Setup".OEM[1].PMC.Machining_Assembly.Starved )
      Coil( "CITI_Logic.OEM_CITI_Logic_Setup".OEM[1].PMC.Machining_Assembly.Wait_1 )
   END_RUNG
   // the same network as SCL:
   "CITI_Logic.OEM_CITI_Logic_Setup".OEM[1].PMC.Machining_Assembly.Wait_1 := "CITI_Logic.zPMC_Configuration".CITI[1].Features.Wait_1 AND "Unit1.EmNodes".oem[1].PMC.Machining_Assembly.Wait_1 AND NOT "CITI_Logic.OEM_CITI_Logic_Setup".OEM[1].PMC.Machining_Assembly.Blocked AND NOT "CITI_Logic.OEM_CITI_Logic_Setup".OEM[1].PMC.Machining_Assembly.Starved;
END_REGION

REGION Network 25: Wait 2 (Check)
   // **Replace the "CITI_Logic_Setup".OEM_TO_COMPLETE Bit with the correct Logic to drive the signal**
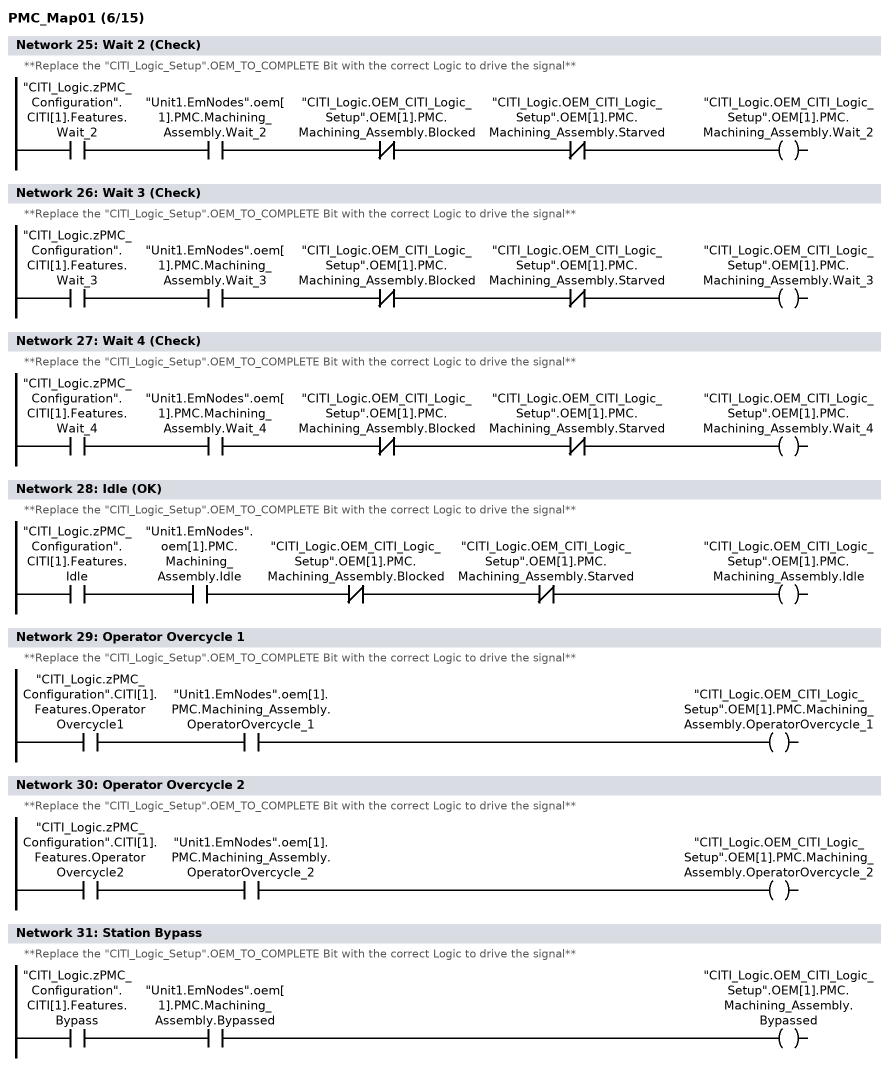
   RUNG wire#powerrail
      Contact( "CITI_Logic.zPMC_Configuration".CITI[1].Features.Wait_2 )
      Contact( "Unit1.EmNodes".oem[1].PMC.Machining_Assembly.Wait_2 )
      I_Contact( "CITI_Logic.OEM_CITI_Logic_Setup".OEM[1].PMC.Machining_Assembly.Blocked )
      I_Contact( "CITI_Logic.OEM_CITI_Logic_Setup".OEM[1].PMC.Machining_Assembly.Starved )
      Coil( "CITI_Logic.OEM_CITI_Logic_Setup".OEM[1].PMC.Machining_Assembly.Wait_2 )
   END_RUNG
   // the same network as SCL:
   "CITI_Logic.OEM_CITI_Logic_Setup".OEM[1].PMC.Machining_Assembly.Wait_2 := "CITI_Logic.zPMC_Configuration".CITI[1].Features.Wait_2 AND "Unit1.EmNodes".oem[1].PMC.Machining_Assembly.Wait_2 AND NOT "CITI_Logic.OEM_CITI_Logic_Setup".OEM[1].PMC.Machining_Assembly.Blocked AND NOT "CITI_Logic.OEM_CITI_Logic_Setup".OEM[1].PMC.Machining_Assembly.Starved;
END_REGION

REGION Network 26: Wait 3 (Check)
   // **Replace the "CITI_Logic_Setup".OEM_TO_COMPLETE Bit with the correct Logic to drive the signal**
   RUNG wire#powerrail
      Contact( "CITI_Logic.zPMC_Configuration".CITI[1].Features.Wait_3 )
      Contact( "Unit1.EmNodes".oem[1].PMC.Machining_Assembly.Wait_3 )
      I_Contact( "CITI_Logic.OEM_CITI_Logic_Setup".OEM[1].PMC.Machining_Assembly.Blocked )
      I_Contact( "CITI_Logic.OEM_CITI_Logic_Setup".OEM[1].PMC.Machining_Assembly.Starved )
      Coil( "CITI_Logic.OEM_CITI_Logic_Setup".OEM[1].PMC.Machining_Assembly.Wait_3 )
   END_RUNG
   // the same network as SCL:
   "CITI_Logic.OEM_CITI_Logic_Setup".OEM[1].PMC.Machining_Assembly.Wait_3 := "CITI_Logic.zPMC_Configuration".CITI[1].Features.Wait_3 AND "Unit1.EmNodes".oem[1].PMC.Machining_Assembly.Wait_3 AND NOT "CITI_Logic.OEM_CITI_Logic_Setup".OEM[1].PMC.Machining_Assembly.Blocked AND NOT "CITI_Logic.OEM_CITI_Logic_Setup".OEM[1].PMC.Machining_Assembly.Starved;
END_REGION

REGION Network 27: Wait 4 (Check)
   // **Replace the "CITI_Logic_Setup".OEM_TO_COMPLETE Bit with the correct Logic to drive the signal**
   RUNG wire#powerrail
      Contact( "CITI_Logic.zPMC_Configuration".CITI[1].Features.Wait_4 )
      Contact( "Unit1.EmNodes".oem[1].PMC.Machining_Assembly.Wait_4 )
      I_Contact( "CITI_Logic.OEM_CITI_Logic_Setup".OEM[1].PMC.Machining_Assembly.Blocked )
      I_Contact( "CITI_Logic.OEM_CITI_Logic_Setup".OEM[1].PMC.Machining_Assembly.Starved )
      Coil( "CITI_Logic.OEM_CITI_Logic_Setup".OEM[1].PMC.Machining_Assembly.Wait_4 )
   END_RUNG
   // the same network as SCL:
   "CITI_Logic.OEM_CITI_Logic_Setup".OEM[1].PMC.Machining_Assembly.Wait_4 := "CITI_Logic.zPMC_Configuration".CITI[1].Features.Wait_4 AND "Unit1.EmNodes".oem[1].PMC.Machining_Assembly.Wait_4 AND NOT "CITI_Logic.OEM_CITI_Logic_Setup".OEM[1].PMC.Machining_Assembly.Blocked AND NOT "CITI_Logic.OEM_CITI_Logic_Setup".OEM[1].PMC.Machining_Assembly.Starved;
END_REGION

REGION Network 28: Idle (OK)
   // **Replace the "CITI_Logic_Setup".OEM_TO_COMPLETE Bit with the correct Logic to drive the signal**
   RUNG wire#powerrail
      Contact( "CITI_Logic.zPMC_Configuration".CITI[1].Features.Idle )
      Contact( "Unit1.EmNodes".oem[1].PMC.Machining_Assembly.Idle )
      I_Contact( "CITI_Logic.OEM_CITI_Logic_Setup".OEM[1].PMC.Machining_Assembly.Blocked )
      I_Contact( "CITI_Logic.OEM_CITI_Logic_Setup".OEM[1].PMC.Machining_Assembly.Starved )
      Coil( "CITI_Logic.OEM_CITI_Logic_Setup".OEM[1].PMC.Machining_Assembly.Idle )
   END_RUNG
   // the same network as SCL:
   "CITI_Logic.OEM_CITI_Logic_Setup".OEM[1].PMC.Machining_Assembly.Idle := "CITI_Logic.zPMC_Configuration".CITI[1].Features.Idle AND "Unit1.EmNodes".oem[1].PMC.Machining_Assembly.Idle AND NOT "CITI_Logic.OEM_CITI_Logic_Setup".OEM[1].PMC.Machining_Assembly.Blocked AND NOT "CITI_Logic.OEM_CITI_Logic_Setup".OEM[1].PMC.Machining_Assembly.Starved;
END_REGION

REGION Network 29: Operator Overcycle 1
   // **Replace the "CITI_Logic_Setup".OEM_TO_COMPLETE Bit with the correct Logic to drive the signal**
   RUNG wire#powerrail
      Contact( "CITI_Logic.zPMC_Configuration".CITI[1].Features.OperatorOvercycle1 )
      Contact( "Unit1.EmNodes".oem[1].PMC.Machining_Assembly.OperatorOvercycle_1 )
      Coil( "CITI_Logic.OEM_CITI_Logic_Setup".OEM[1].PMC.Machining_Assembly.OperatorOvercycle_1 )
   END_RUNG
   // the same network as SCL:
   "CITI_Logic.OEM_CITI_Logic_Setup".OEM[1].PMC.Machining_Assembly.OperatorOvercycle_1 := "CITI_Logic.zPMC_Configuration".CITI[1].Features.OperatorOvercycle1 AND "Unit1.EmNodes".oem[1].PMC.Machining_Assembly.OperatorOvercycle_1;
END_REGION

REGION Network 30: Operator Overcycle 2
   // **Replace the "CITI_Logic_Setup".OEM_TO_COMPLETE Bit with the correct Logic to drive the signal**
   RUNG wire#powerrail
      Contact( "CITI_Logic.zPMC_Configuration".CITI[1].Features.OperatorOvercycle2 )
      Contact( "Unit1.EmNodes".oem[1].PMC.Machining_Assembly.OperatorOvercycle_2 )
      Coil( "CITI_Logic.OEM_CITI_Logic_Setup".OEM[1].PMC.Machining_Assembly.OperatorOvercycle_2 )
   END_RUNG
   // the same network as SCL:
   "CITI_Logic.OEM_CITI_Logic_Setup".OEM[1].PMC.Machining_Assembly.OperatorOvercycle_2 := "CITI_Logic.zPMC_Configuration".CITI[1].Features.OperatorOvercycle2 AND "Unit1.EmNodes".oem[1].PMC.Machining_Assembly.OperatorOvercycle_2;
END_REGION

REGION Network 31: Station Bypass
   // **Replace the "CITI_Logic_Setup".OEM_TO_COMPLETE Bit with the correct Logic to drive the signal**
   RUNG wire#powerrail
      Contact( "CITI_Logic.zPMC_Configuration".CITI[1].Features.Bypass )
      Contact( "Unit1.EmNodes".oem[1].PMC.Machining_Assembly.Bypassed )
      Coil( "CITI_Logic.OEM_CITI_Logic_Setup".OEM[1].PMC.Machining_Assembly.Bypassed )
   END_RUNG
   // the same network as SCL:
   "CITI_Logic.OEM_CITI_Logic_Setup".OEM[1].PMC.Machining_Assembly.Bypassed := "CITI_Logic.zPMC_Configuration".CITI[1].Features.Bypass AND "Unit1.EmNodes".oem[1].PMC.Machining_Assembly.Bypassed;
END_REGION

REGION Network 32: Good Count Trigger
   // **Replace the "CITI_Logic_Setup".OEM_TO_COMPLETE Bit with the correct Logic to drive the signal**
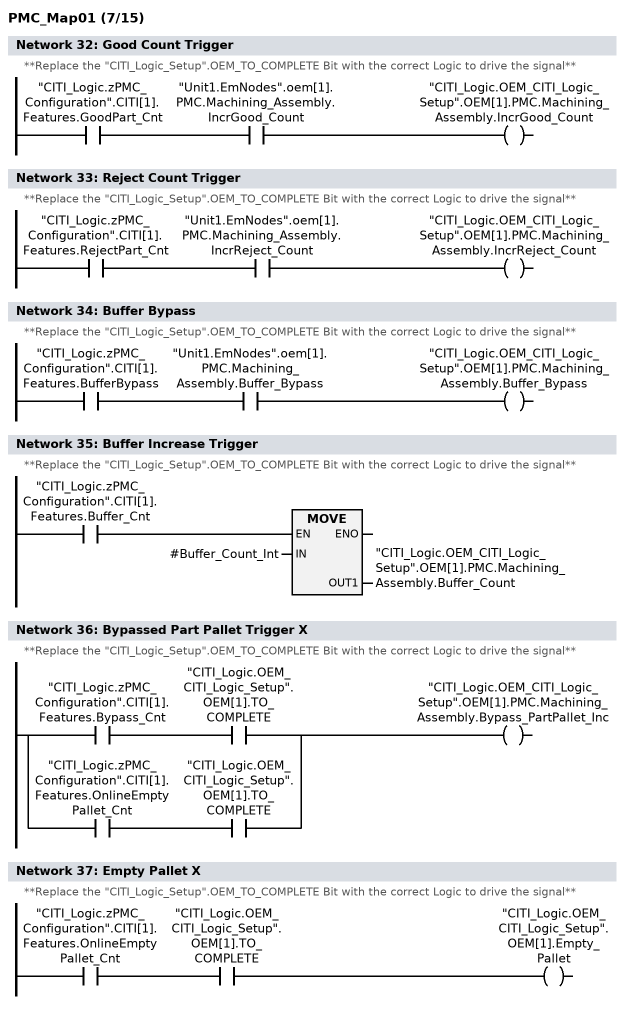
   RUNG wire#powerrail
      Contact( "CITI_Logic.zPMC_Configuration".CITI[1].Features.GoodPart_Cnt )
      Contact( "Unit1.EmNodes".oem[1].PMC.Machining_Assembly.IncrGood_Count )
      Coil( "CITI_Logic.OEM_CITI_Logic_Setup".OEM[1].PMC.Machining_Assembly.IncrGood_Count )
   END_RUNG
   // the same network as SCL:
   "CITI_Logic.OEM_CITI_Logic_Setup".OEM[1].PMC.Machining_Assembly.IncrGood_Count := "CITI_Logic.zPMC_Configuration".CITI[1].Features.GoodPart_Cnt AND "Unit1.EmNodes".oem[1].PMC.Machining_Assembly.IncrGood_Count;
END_REGION

REGION Network 33: Reject Count Trigger
   // **Replace the "CITI_Logic_Setup".OEM_TO_COMPLETE Bit with the correct Logic to drive the signal**
   RUNG wire#powerrail
      Contact( "CITI_Logic.zPMC_Configuration".CITI[1].Features.RejectPart_Cnt )
      Contact( "Unit1.EmNodes".oem[1].PMC.Machining_Assembly.IncrReject_Count )
      Coil( "CITI_Logic.OEM_CITI_Logic_Setup".OEM[1].PMC.Machining_Assembly.IncrReject_Count )
   END_RUNG
   // the same network as SCL:
   "CITI_Logic.OEM_CITI_Logic_Setup".OEM[1].PMC.Machining_Assembly.IncrReject_Count := "CITI_Logic.zPMC_Configuration".CITI[1].Features.RejectPart_Cnt AND "Unit1.EmNodes".oem[1].PMC.Machining_Assembly.IncrReject_Count;
END_REGION

REGION Network 34: Buffer Bypass
   // **Replace the "CITI_Logic_Setup".OEM_TO_COMPLETE Bit with the correct Logic to drive the signal**
   RUNG wire#powerrail
      Contact( "CITI_Logic.zPMC_Configuration".CITI[1].Features.BufferBypass )
      Contact( "Unit1.EmNodes".oem[1].PMC.Machining_Assembly.Buffer_Bypass )
      Coil( "CITI_Logic.OEM_CITI_Logic_Setup".OEM[1].PMC.Machining_Assembly.Buffer_Bypass )
   END_RUNG
   // the same network as SCL:
   "CITI_Logic.OEM_CITI_Logic_Setup".OEM[1].PMC.Machining_Assembly.Buffer_Bypass := "CITI_Logic.zPMC_Configuration".CITI[1].Features.BufferBypass AND "Unit1.EmNodes".oem[1].PMC.Machining_Assembly.Buffer_Bypass;
END_REGION

REGION Network 35: Buffer Increase Trigger
   // **Replace the "CITI_Logic_Setup".OEM_TO_COMPLETE Bit with the correct Logic to drive the signal**
   RUNG wire#powerrail
      Contact( "CITI_Logic.zPMC_Configuration".CITI[1].Features.Buffer_Cnt )
      Move(in := #Buffer_Count_Int, out1 => "CITI_Logic.OEM_CITI_Logic_Setup".OEM[1].PMC.Machining_Assembly.Buffer_Count)
   END_RUNG
   // the same network as SCL:
   IF "CITI_Logic.zPMC_Configuration".CITI[1].Features.Buffer_Cnt THEN
       "CITI_Logic.OEM_CITI_Logic_Setup".OEM[1].PMC.Machining_Assembly.Buffer_Count := #Buffer_Count_Int;
   END_IF;
END_REGION

REGION Network 36: Bypassed Part Pallet Trigger X
   // **Replace the "CITI_Logic_Setup".OEM_TO_COMPLETE Bit with the correct Logic to drive the signal**
   RUNG wire#powerrail
      Contact( "CITI_Logic.zPMC_Configuration".CITI[1].Features.Bypass_Cnt )
      Contact( "CITI_Logic.OEM_CITI_Logic_Setup".OEM[1].TO_COMPLETE )
      wire#w1
      Coil( "CITI_Logic.OEM_CITI_Logic_Setup".OEM[1].PMC.Machining_Assembly.Bypass_PartPallet_Inc )
   END_RUNG
   RUNG wire#powerrail
      Contact( "CITI_Logic.zPMC_Configuration".CITI[1].Features.OnlineEmptyPallet_Cnt )
      Contact( "CITI_Logic.OEM_CITI_Logic_Setup".OEM[1].TO_COMPLETE )
   END_RUNG wire#w1
   // the same network as SCL:
   "CITI_Logic.OEM_CITI_Logic_Setup".OEM[1].PMC.Machining_Assembly.Bypass_PartPallet_Inc := ("CITI_Logic.zPMC_Configuration".CITI[1].Features.Bypass_Cnt AND "CITI_Logic.OEM_CITI_Logic_Setup".OEM[1].TO_COMPLETE) OR ("CITI_Logic.zPMC_Configuration".CITI[1].Features.OnlineEmptyPallet_Cnt AND "CITI_Logic.OEM_CITI_Logic_Setup".OEM[1].TO_COMPLETE);
END_REGION

REGION Network 37: Empty Pallet X
   // **Replace the "CITI_Logic_Setup".OEM_TO_COMPLETE Bit with the correct Logic to drive the signal**
   RUNG wire#powerrail
      Contact( "CITI_Logic.zPMC_Configuration".CITI[1].Features.OnlineEmptyPallet_Cnt )
      Contact( "CITI_Logic.OEM_CITI_Logic_Setup".OEM[1].TO_COMPLETE )
      Coil( "CITI_Logic.OEM_CITI_Logic_Setup".OEM[1].Empty_Pallet )
   END_RUNG
   // the same network as SCL:
   "CITI_Logic.OEM_CITI_Logic_Setup".OEM[1].Empty_Pallet := "CITI_Logic.zPMC_Configuration".CITI[1].Features.OnlineEmptyPallet_Cnt AND "CITI_Logic.OEM_CITI_Logic_Setup".OEM[1].TO_COMPLETE;
END_REGION

REGION Network 38: PUN, GM Part Number, and Optional Data Copy
   // **Replace the "CITI_Logic_Setup".OEM_TO_COMPLETE Bit with the correct Logic to drive the signal**
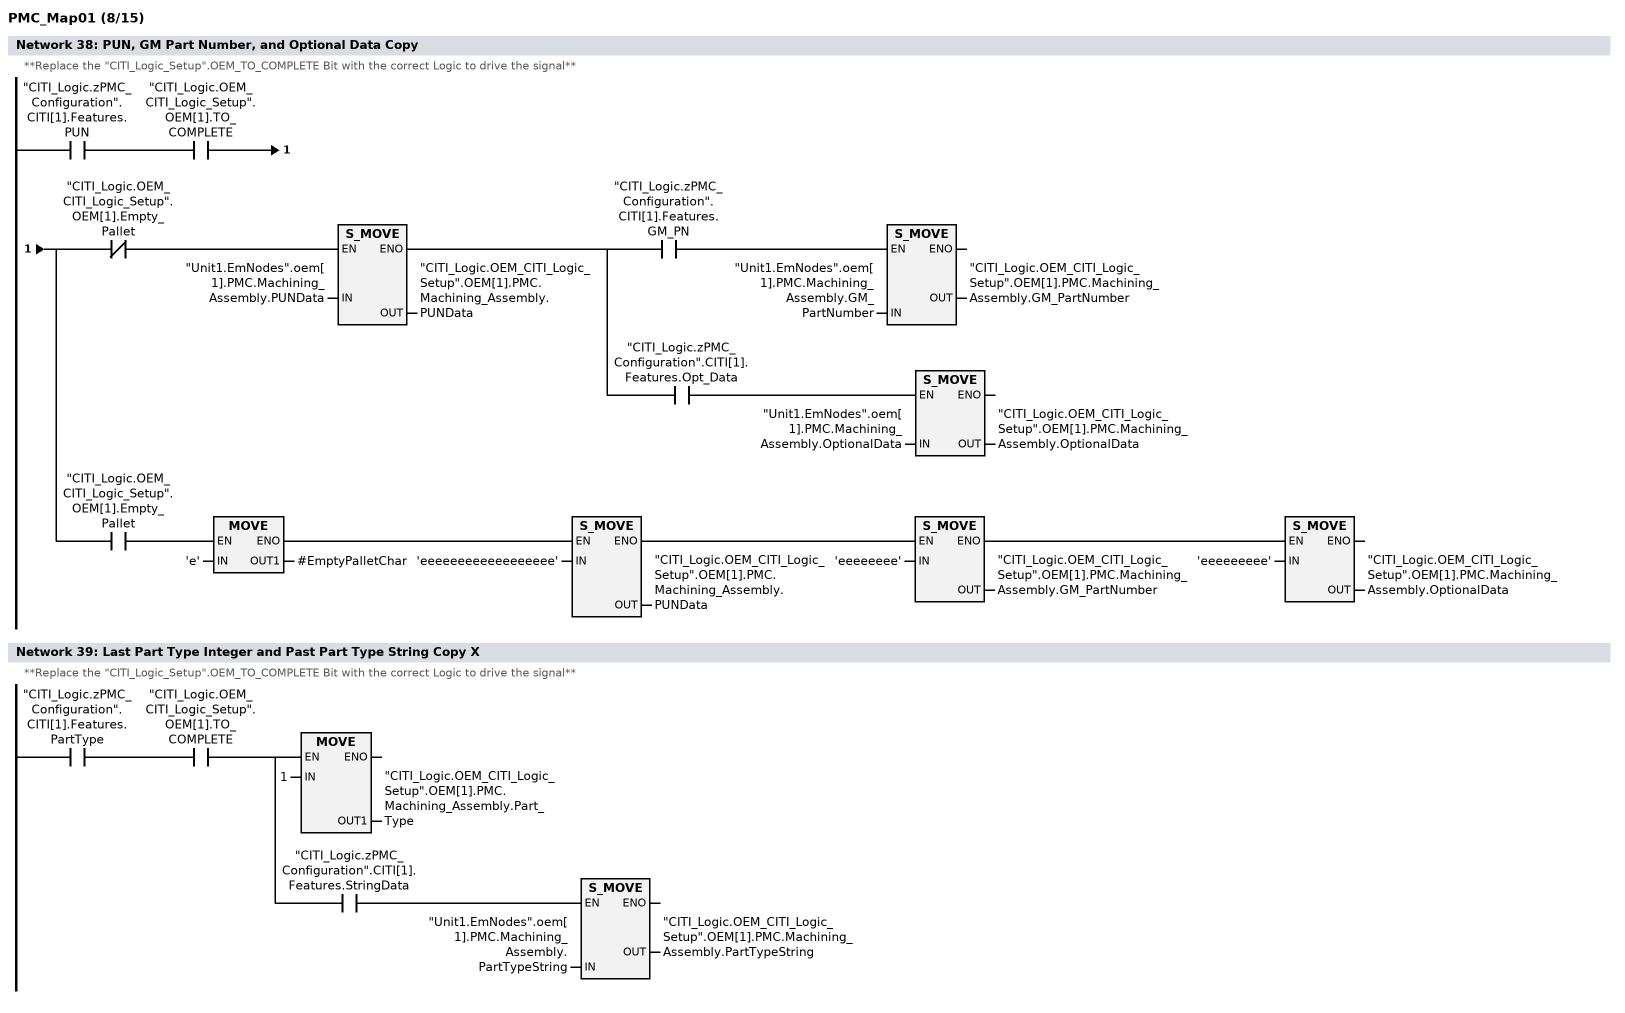
   RUNG wire#powerrail
      Contact( "CITI_Logic.zPMC_Configuration".CITI[1].Features.PUN )
      Contact( "CITI_Logic.OEM_CITI_Logic_Setup".OEM[1].TO_COMPLETE )
      wire#w1
      I_Contact( "CITI_Logic.OEM_CITI_Logic_Setup".OEM[1].Empty_Pallet )
      S_Move(in := "Unit1.EmNodes".oem[1].PMC.Machining_Assembly.PUNData, out => "CITI_Logic.OEM_CITI_Logic_Setup".OEM[1].PMC.Machining_Assembly.PUNData)
      wire#w2
      Contact( "CITI_Logic.zPMC_Configuration".CITI[1].Features.GM_PN )
      S_Move(in := "Unit1.EmNodes".oem[1].PMC.Machining_Assembly.GM_PartNumber, out => "CITI_Logic.OEM_CITI_Logic_Setup".OEM[1].PMC.Machining_Assembly.GM_PartNumber)
   END_RUNG
   RUNG wire#w2
      Contact( "CITI_Logic.zPMC_Configuration".CITI[1].Features.Opt_Data )
      S_Move(in := "Unit1.EmNodes".oem[1].PMC.Machining_Assembly.OptionalData, out => "CITI_Logic.OEM_CITI_Logic_Setup".OEM[1].PMC.Machining_Assembly.OptionalData)
   END_RUNG
   RUNG wire#w1
      Contact( "CITI_Logic.OEM_CITI_Logic_Setup".OEM[1].Empty_Pallet )
      { S7_GenerateENO := "TRUE" } Move(in := 'e', out1 => #EmptyPalletChar)
      S_Move(in := 'eeeeeeeeeeeeeeeeee', out => "CITI_Logic.OEM_CITI_Logic_Setup".OEM[1].PMC.Machining_Assembly.PUNData)
      S_Move(in := 'eeeeeeee', out => "CITI_Logic.OEM_CITI_Logic_Setup".OEM[1].PMC.Machining_Assembly.GM_PartNumber)
      S_Move(in := 'eeeeeeeee', out => "CITI_Logic.OEM_CITI_Logic_Setup".OEM[1].PMC.Machining_Assembly.OptionalData)
   END_RUNG
   // the same network as SCL:
   // ENO of a box is taken as its EN; it also drops when the box reports an error
   #_w1 := "CITI_Logic.zPMC_Configuration".CITI[1].Features.PUN AND "CITI_Logic.OEM_CITI_Logic_Setup".OEM[1].TO_COMPLETE;
   #_w2 := #_w1 AND NOT "CITI_Logic.OEM_CITI_Logic_Setup".OEM[1].Empty_Pallet;
   IF #_w2 THEN
       "CITI_Logic.OEM_CITI_Logic_Setup".OEM[1].PMC.Machining_Assembly.PUNData := "Unit1.EmNodes".oem[1].PMC.Machining_Assembly.PUNData;
   END_IF;
   IF #_w2 AND "CITI_Logic.zPMC_Configuration".CITI[1].Features.GM_PN THEN
       "CITI_Logic.OEM_CITI_Logic_Setup".OEM[1].PMC.Machining_Assembly.GM_PartNumber := "Unit1.EmNodes".oem[1].PMC.Machining_Assembly.GM_PartNumber;
   END_IF;
   IF #_w2 AND "CITI_Logic.zPMC_Configuration".CITI[1].Features.Opt_Data THEN
       "CITI_Logic.OEM_CITI_Logic_Setup".OEM[1].PMC.Machining_Assembly.OptionalData := "Unit1.EmNodes".oem[1].PMC.Machining_Assembly.OptionalData;
   END_IF;
   IF #_w1 AND "CITI_Logic.OEM_CITI_Logic_Setup".OEM[1].Empty_Pallet THEN #EmptyPalletChar := 'e'; END_IF;
   #_w3 := #_w1 AND "CITI_Logic.OEM_CITI_Logic_Setup".OEM[1].Empty_Pallet;
   IF #_w3 THEN
       "CITI_Logic.OEM_CITI_Logic_Setup".OEM[1].PMC.Machining_Assembly.PUNData := 'eeeeeeeeeeeeeeeeee';
       "CITI_Logic.OEM_CITI_Logic_Setup".OEM[1].PMC.Machining_Assembly.GM_PartNumber := 'eeeeeeee';
       "CITI_Logic.OEM_CITI_Logic_Setup".OEM[1].PMC.Machining_Assembly.OptionalData := 'eeeeeeeee';
   END_IF;
END_REGION

REGION Network 39: Last Part Type Integer and Past Part Type String Copy X
   // **Replace the "CITI_Logic_Setup".OEM_TO_COMPLETE Bit with the correct Logic to drive the signal**
   RUNG wire#powerrail
      Contact( "CITI_Logic.zPMC_Configuration".CITI[1].Features.PartType )
      Contact( "CITI_Logic.OEM_CITI_Logic_Setup".OEM[1].TO_COMPLETE )
      wire#w1
      Move(in := 1, out1 => "CITI_Logic.OEM_CITI_Logic_Setup".OEM[1].PMC.Machining_Assembly.Part_Type)
   END_RUNG
   RUNG wire#w1
      Contact( "CITI_Logic.zPMC_Configuration".CITI[1].Features.StringData )
      S_Move(in := "Unit1.EmNodes".oem[1].PMC.Machining_Assembly.PartTypeString, out => "CITI_Logic.OEM_CITI_Logic_Setup".OEM[1].PMC.Machining_Assembly.PartTypeString)
   END_RUNG
   // the same network as SCL:
   #_w1 := "CITI_Logic.zPMC_Configuration".CITI[1].Features.PartType AND "CITI_Logic.OEM_CITI_Logic_Setup".OEM[1].TO_COMPLETE;
   IF #_w1 THEN "CITI_Logic.OEM_CITI_Logic_Setup".OEM[1].PMC.Machining_Assembly.Part_Type := 1; END_IF;
   IF #_w1 AND "CITI_Logic.zPMC_Configuration".CITI[1].Features.StringData THEN
       "CITI_Logic.OEM_CITI_Logic_Setup".OEM[1].PMC.Machining_Assembly.PartTypeString := "Unit1.EmNodes".oem[1].PMC.Machining_Assembly.PartTypeString;
   END_IF;
END_REGION

REGION Network 40: FTQ PUN, String, and FTQ Integer Copy (N/A)
   // **Replace the "CITI_Logic_Setup".OEM_TO_COMPLETE Bit with the correct Logic to drive the signal**
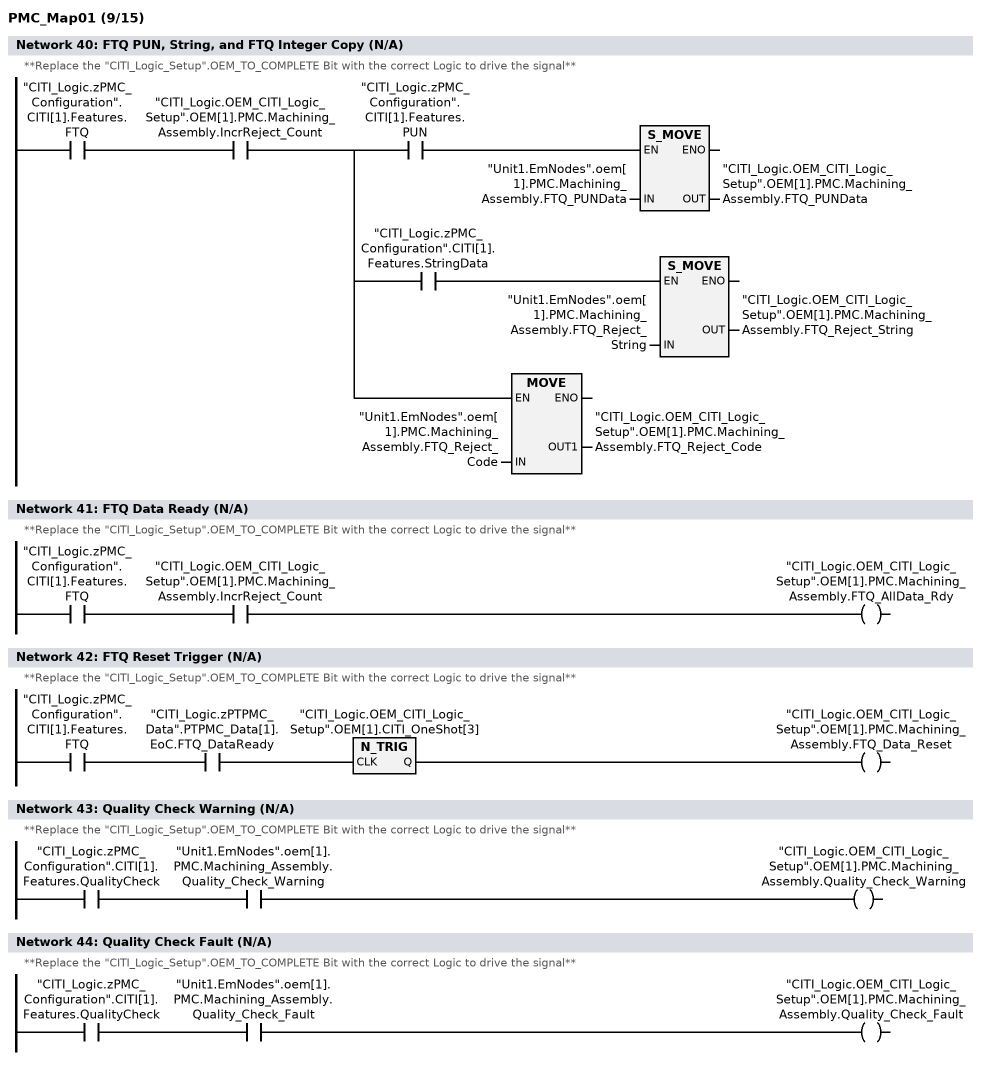
   RUNG wire#powerrail
      Contact( "CITI_Logic.zPMC_Configuration".CITI[1].Features.FTQ )
      Contact( "CITI_Logic.OEM_CITI_Logic_Setup".OEM[1].PMC.Machining_Assembly.IncrReject_Count )
      wire#w1
      Contact( "CITI_Logic.zPMC_Configuration".CITI[1].Features.PUN )
      S_Move(in := "Unit1.EmNodes".oem[1].PMC.Machining_Assembly.FTQ_PUNData, out => "CITI_Logic.OEM_CITI_Logic_Setup".OEM[1].PMC.Machining_Assembly.FTQ_PUNData)
   END_RUNG
   RUNG wire#w1
      Contact( "CITI_Logic.zPMC_Configuration".CITI[1].Features.StringData )
      S_Move(in := "Unit1.EmNodes".oem[1].PMC.Machining_Assembly.FTQ_Reject_String, out => "CITI_Logic.OEM_CITI_Logic_Setup".OEM[1].PMC.Machining_Assembly.FTQ_Reject_String)
   END_RUNG
   RUNG wire#w1
      Move(in := "Unit1.EmNodes".oem[1].PMC.Machining_Assembly.FTQ_Reject_Code, out1 => "CITI_Logic.OEM_CITI_Logic_Setup".OEM[1].PMC.Machining_Assembly.FTQ_Reject_Code)
   END_RUNG
   // the same network as SCL:
   #_w1 := "CITI_Logic.zPMC_Configuration".CITI[1].Features.FTQ AND "CITI_Logic.OEM_CITI_Logic_Setup".OEM[1].PMC.Machining_Assembly.IncrReject_Count;
   IF #_w1 AND "CITI_Logic.zPMC_Configuration".CITI[1].Features.PUN THEN
       "CITI_Logic.OEM_CITI_Logic_Setup".OEM[1].PMC.Machining_Assembly.FTQ_PUNData := "Unit1.EmNodes".oem[1].PMC.Machining_Assembly.FTQ_PUNData;
   END_IF;
   IF #_w1 AND "CITI_Logic.zPMC_Configuration".CITI[1].Features.StringData THEN
       "CITI_Logic.OEM_CITI_Logic_Setup".OEM[1].PMC.Machining_Assembly.FTQ_Reject_String := "Unit1.EmNodes".oem[1].PMC.Machining_Assembly.FTQ_Reject_String;
   END_IF;
   IF #_w1 THEN
       "CITI_Logic.OEM_CITI_Logic_Setup".OEM[1].PMC.Machining_Assembly.FTQ_Reject_Code := "Unit1.EmNodes".oem[1].PMC.Machining_Assembly.FTQ_Reject_Code;
   END_IF;
END_REGION

REGION Network 41: FTQ Data Ready (N/A)
   // **Replace the "CITI_Logic_Setup".OEM_TO_COMPLETE Bit with the correct Logic to drive the signal**
   RUNG wire#powerrail
      Contact( "CITI_Logic.zPMC_Configuration".CITI[1].Features.FTQ )
      Contact( "CITI_Logic.OEM_CITI_Logic_Setup".OEM[1].PMC.Machining_Assembly.IncrReject_Count )
      Coil( "CITI_Logic.OEM_CITI_Logic_Setup".OEM[1].PMC.Machining_Assembly.FTQ_AllData_Rdy )
   END_RUNG
   // the same network as SCL:
   "CITI_Logic.OEM_CITI_Logic_Setup".OEM[1].PMC.Machining_Assembly.FTQ_AllData_Rdy := "CITI_Logic.zPMC_Configuration".CITI[1].Features.FTQ AND "CITI_Logic.OEM_CITI_Logic_Setup".OEM[1].PMC.Machining_Assembly.IncrReject_Count;
END_REGION

REGION Network 42: FTQ Reset Trigger (N/A)
   // **Replace the "CITI_Logic_Setup".OEM_TO_COMPLETE Bit with the correct Logic to drive the signal**
   RUNG wire#powerrail
      Contact( "CITI_Logic.zPMC_Configuration".CITI[1].Features.FTQ )
      Contact( "CITI_Logic.zPTPMC_Data".PTPMC_Data[1].EoC.FTQ_DataReady )
      N_Trig( "CITI_Logic.OEM_CITI_Logic_Setup".OEM[1].CITI_OneShot[3] )
      Coil( "CITI_Logic.OEM_CITI_Logic_Setup".OEM[1].PMC.Machining_Assembly.FTQ_Data_Reset )
   END_RUNG
   // the same network as SCL:
   #_w1 := "CITI_Logic.zPMC_Configuration".CITI[1].Features.FTQ AND "CITI_Logic.zPTPMC_Data".PTPMC_Data[1].EoC.FTQ_DataReady;
   #_w2 := NOT #_w1 AND "CITI_Logic.OEM_CITI_Logic_Setup".OEM[1].CITI_OneShot[3];   // falling edge
   "CITI_Logic.OEM_CITI_Logic_Setup".OEM[1].CITI_OneShot[3] := #_w1;
   "CITI_Logic.OEM_CITI_Logic_Setup".OEM[1].PMC.Machining_Assembly.FTQ_Data_Reset := #_w2;
END_REGION

REGION Network 43: Quality Check Warning (N/A)
   // **Replace the "CITI_Logic_Setup".OEM_TO_COMPLETE Bit with the correct Logic to drive the signal**
   RUNG wire#powerrail
      Contact( "CITI_Logic.zPMC_Configuration".CITI[1].Features.QualityCheck )
      Contact( "Unit1.EmNodes".oem[1].PMC.Machining_Assembly.Quality_Check_Warning )
      Coil( "CITI_Logic.OEM_CITI_Logic_Setup".OEM[1].PMC.Machining_Assembly.Quality_Check_Warning )
   END_RUNG
   // the same network as SCL:
   "CITI_Logic.OEM_CITI_Logic_Setup".OEM[1].PMC.Machining_Assembly.Quality_Check_Warning := "CITI_Logic.zPMC_Configuration".CITI[1].Features.QualityCheck AND "Unit1.EmNodes".oem[1].PMC.Machining_Assembly.Quality_Check_Warning;
END_REGION

REGION Network 44: Quality Check Fault (N/A)
   // **Replace the "CITI_Logic_Setup".OEM_TO_COMPLETE Bit with the correct Logic to drive the signal**
   RUNG wire#powerrail
      Contact( "CITI_Logic.zPMC_Configuration".CITI[1].Features.QualityCheck )
      Contact( "Unit1.EmNodes".oem[1].PMC.Machining_Assembly.Quality_Check_Fault )
      Coil( "CITI_Logic.OEM_CITI_Logic_Setup".OEM[1].PMC.Machining_Assembly.Quality_Check_Fault )
   END_RUNG
   // the same network as SCL:
   "CITI_Logic.OEM_CITI_Logic_Setup".OEM[1].PMC.Machining_Assembly.Quality_Check_Fault := "CITI_Logic.zPMC_Configuration".CITI[1].Features.QualityCheck AND "Unit1.EmNodes".oem[1].PMC.Machining_Assembly.Quality_Check_Fault;
END_REGION

REGION Network 45: Quality Check Acknowledge (N/A)
   // **Replace the "CITI_Logic_Setup".OEM_TO_COMPLETE Bit with the correct Logic to drive the signal**
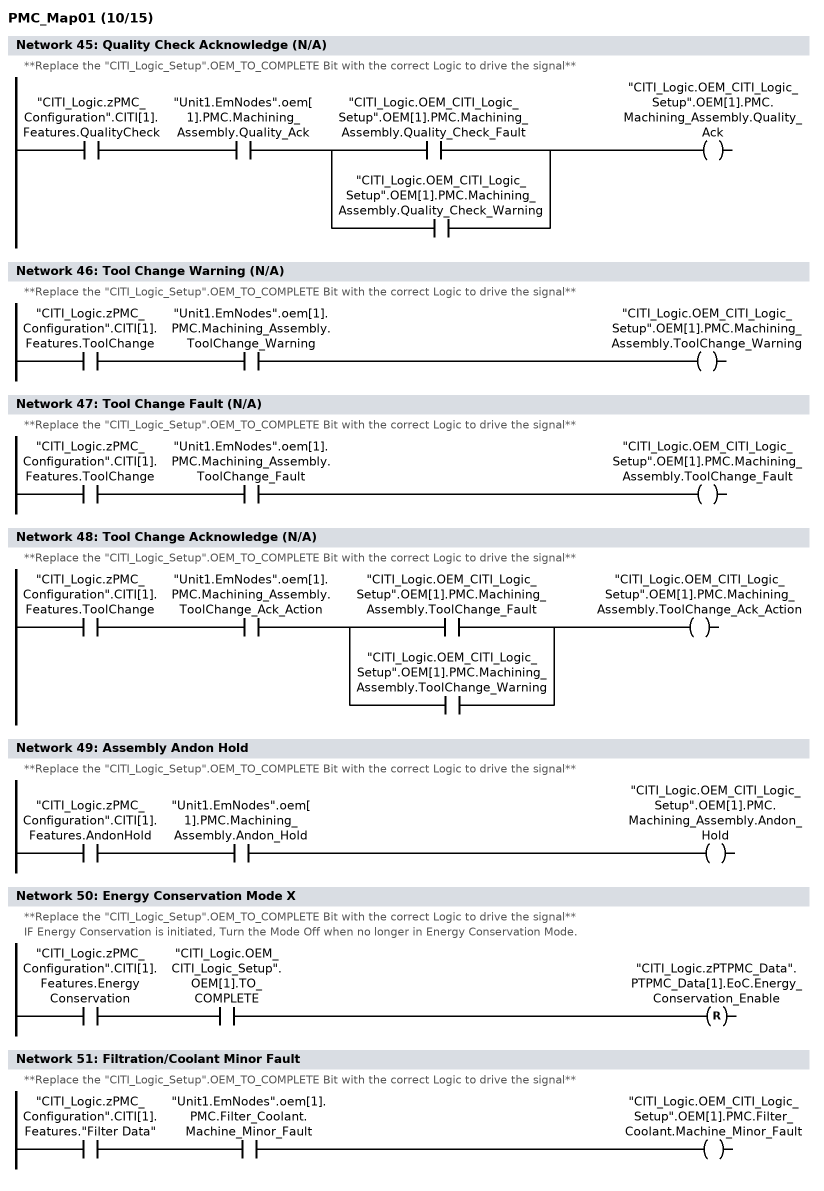
   RUNG wire#powerrail
      Contact( "CITI_Logic.zPMC_Configuration".CITI[1].Features.QualityCheck )
      Contact( "Unit1.EmNodes".oem[1].PMC.Machining_Assembly.Quality_Ack )
      wire#w1
      Contact( "CITI_Logic.OEM_CITI_Logic_Setup".OEM[1].PMC.Machining_Assembly.Quality_Check_Fault )
      wire#w2
      Coil( "CITI_Logic.OEM_CITI_Logic_Setup".OEM[1].PMC.Machining_Assembly.Quality_Ack )
   END_RUNG
   RUNG wire#w1
      Contact( "CITI_Logic.OEM_CITI_Logic_Setup".OEM[1].PMC.Machining_Assembly.Quality_Check_Warning )
   END_RUNG wire#w2
   // the same network as SCL:
   "CITI_Logic.OEM_CITI_Logic_Setup".OEM[1].PMC.Machining_Assembly.Quality_Ack := "CITI_Logic.zPMC_Configuration".CITI[1].Features.QualityCheck AND "Unit1.EmNodes".oem[1].PMC.Machining_Assembly.Quality_Ack AND ("CITI_Logic.OEM_CITI_Logic_Setup".OEM[1].PMC.Machining_Assembly.Quality_Check_Fault OR "CITI_Logic.OEM_CITI_Logic_Setup".OEM[1].PMC.Machining_Assembly.Quality_Check_Warning);
END_REGION

REGION Network 46: Tool Change Warning (N/A)
   // **Replace the "CITI_Logic_Setup".OEM_TO_COMPLETE Bit with the correct Logic to drive the signal**
   RUNG wire#powerrail
      Contact( "CITI_Logic.zPMC_Configuration".CITI[1].Features.ToolChange )
      Contact( "Unit1.EmNodes".oem[1].PMC.Machining_Assembly.ToolChange_Warning )
      Coil( "CITI_Logic.OEM_CITI_Logic_Setup".OEM[1].PMC.Machining_Assembly.ToolChange_Warning )
   END_RUNG
   // the same network as SCL:
   "CITI_Logic.OEM_CITI_Logic_Setup".OEM[1].PMC.Machining_Assembly.ToolChange_Warning := "CITI_Logic.zPMC_Configuration".CITI[1].Features.ToolChange AND "Unit1.EmNodes".oem[1].PMC.Machining_Assembly.ToolChange_Warning;
END_REGION

REGION Network 47: Tool Change Fault (N/A)
   // **Replace the "CITI_Logic_Setup".OEM_TO_COMPLETE Bit with the correct Logic to drive the signal**
   RUNG wire#powerrail
      Contact( "CITI_Logic.zPMC_Configuration".CITI[1].Features.ToolChange )
      Contact( "Unit1.EmNodes".oem[1].PMC.Machining_Assembly.ToolChange_Fault )
      Coil( "CITI_Logic.OEM_CITI_Logic_Setup".OEM[1].PMC.Machining_Assembly.ToolChange_Fault )
   END_RUNG
   // the same network as SCL:
   "CITI_Logic.OEM_CITI_Logic_Setup".OEM[1].PMC.Machining_Assembly.ToolChange_Fault := "CITI_Logic.zPMC_Configuration".CITI[1].Features.ToolChange AND "Unit1.EmNodes".oem[1].PMC.Machining_Assembly.ToolChange_Fault;
END_REGION

REGION Network 48: Tool Change Acknowledge (N/A)
   // **Replace the "CITI_Logic_Setup".OEM_TO_COMPLETE Bit with the correct Logic to drive the signal**
   RUNG wire#powerrail
      Contact( "CITI_Logic.zPMC_Configuration".CITI[1].Features.ToolChange )
      Contact( "Unit1.EmNodes".oem[1].PMC.Machining_Assembly.ToolChange_Ack_Action )
      wire#w1
      Contact( "CITI_Logic.OEM_CITI_Logic_Setup".OEM[1].PMC.Machining_Assembly.ToolChange_Fault )
      wire#w2
      Coil( "CITI_Logic.OEM_CITI_Logic_Setup".OEM[1].PMC.Machining_Assembly.ToolChange_Ack_Action )
   END_RUNG
   RUNG wire#w1
      Contact( "CITI_Logic.OEM_CITI_Logic_Setup".OEM[1].PMC.Machining_Assembly.ToolChange_Warning )
   END_RUNG wire#w2
   // the same network as SCL:
   "CITI_Logic.OEM_CITI_Logic_Setup".OEM[1].PMC.Machining_Assembly.ToolChange_Ack_Action := "CITI_Logic.zPMC_Configuration".CITI[1].Features.ToolChange AND "Unit1.EmNodes".oem[1].PMC.Machining_Assembly.ToolChange_Ack_Action AND ("CITI_Logic.OEM_CITI_Logic_Setup".OEM[1].PMC.Machining_Assembly.ToolChange_Fault OR "CITI_Logic.OEM_CITI_Logic_Setup".OEM[1].PMC.Machining_Assembly.ToolChange_Warning);
END_REGION

REGION Network 49: Assembly Andon Hold
   // **Replace the "CITI_Logic_Setup".OEM_TO_COMPLETE Bit with the correct Logic to drive the signal**
   RUNG wire#powerrail
      Contact( "CITI_Logic.zPMC_Configuration".CITI[1].Features.AndonHold )
      Contact( "Unit1.EmNodes".oem[1].PMC.Machining_Assembly.Andon_Hold )
      Coil( "CITI_Logic.OEM_CITI_Logic_Setup".OEM[1].PMC.Machining_Assembly.Andon_Hold )
   END_RUNG
   // the same network as SCL:
   "CITI_Logic.OEM_CITI_Logic_Setup".OEM[1].PMC.Machining_Assembly.Andon_Hold := "CITI_Logic.zPMC_Configuration".CITI[1].Features.AndonHold AND "Unit1.EmNodes".oem[1].PMC.Machining_Assembly.Andon_Hold;
END_REGION

REGION Network 50: Energy Conservation Mode X
   // **Replace the "CITI_Logic_Setup".OEM_TO_COMPLETE Bit with the correct Logic to drive the signal**
   // 
   // IF Energy Conservation is initiated, Turn the Mode Off when no longer in Energy Conservation Mode.
   RUNG wire#powerrail
      Contact( "CITI_Logic.zPMC_Configuration".CITI[1].Features.EnergyConservation )
      Contact( "CITI_Logic.OEM_CITI_Logic_Setup".OEM[1].TO_COMPLETE )
      R_Coil( "CITI_Logic.zPTPMC_Data".PTPMC_Data[1].EoC.Energy_Conservation_Enable )
   END_RUNG
   // the same network as SCL:
   IF "CITI_Logic.zPMC_Configuration".CITI[1].Features.EnergyConservation AND "CITI_Logic.OEM_CITI_Logic_Setup".OEM[1].TO_COMPLETE THEN
       "CITI_Logic.zPTPMC_Data".PTPMC_Data[1].EoC.Energy_Conservation_Enable := FALSE;
   END_IF;
END_REGION

REGION Network 51: Filtration/Coolant Minor Fault
   // **Replace the "CITI_Logic_Setup".OEM_TO_COMPLETE Bit with the correct Logic to drive the signal**
   RUNG wire#powerrail
      Contact( "CITI_Logic.zPMC_Configuration".CITI[1].Features."Filter Data" )
      Contact( "Unit1.EmNodes".oem[1].PMC.Filter_Coolant.Machine_Minor_Fault )
      Coil( "CITI_Logic.OEM_CITI_Logic_Setup".OEM[1].PMC.Filter_Coolant.Machine_Minor_Fault )
   END_RUNG
   // the same network as SCL:
   "CITI_Logic.OEM_CITI_Logic_Setup".OEM[1].PMC.Filter_Coolant.Machine_Minor_Fault := "CITI_Logic.zPMC_Configuration".CITI[1].Features."Filter Data" AND "Unit1.EmNodes".oem[1].PMC.Filter_Coolant.Machine_Minor_Fault;
END_REGION

REGION Network 52: Filtration/Coolant Current Temperature and Numeric Quantities
   // **Replace the "CITI_Logic_Setup".OEM_TO_COMPLETE_INT" with the correct Logic to drive the signal**
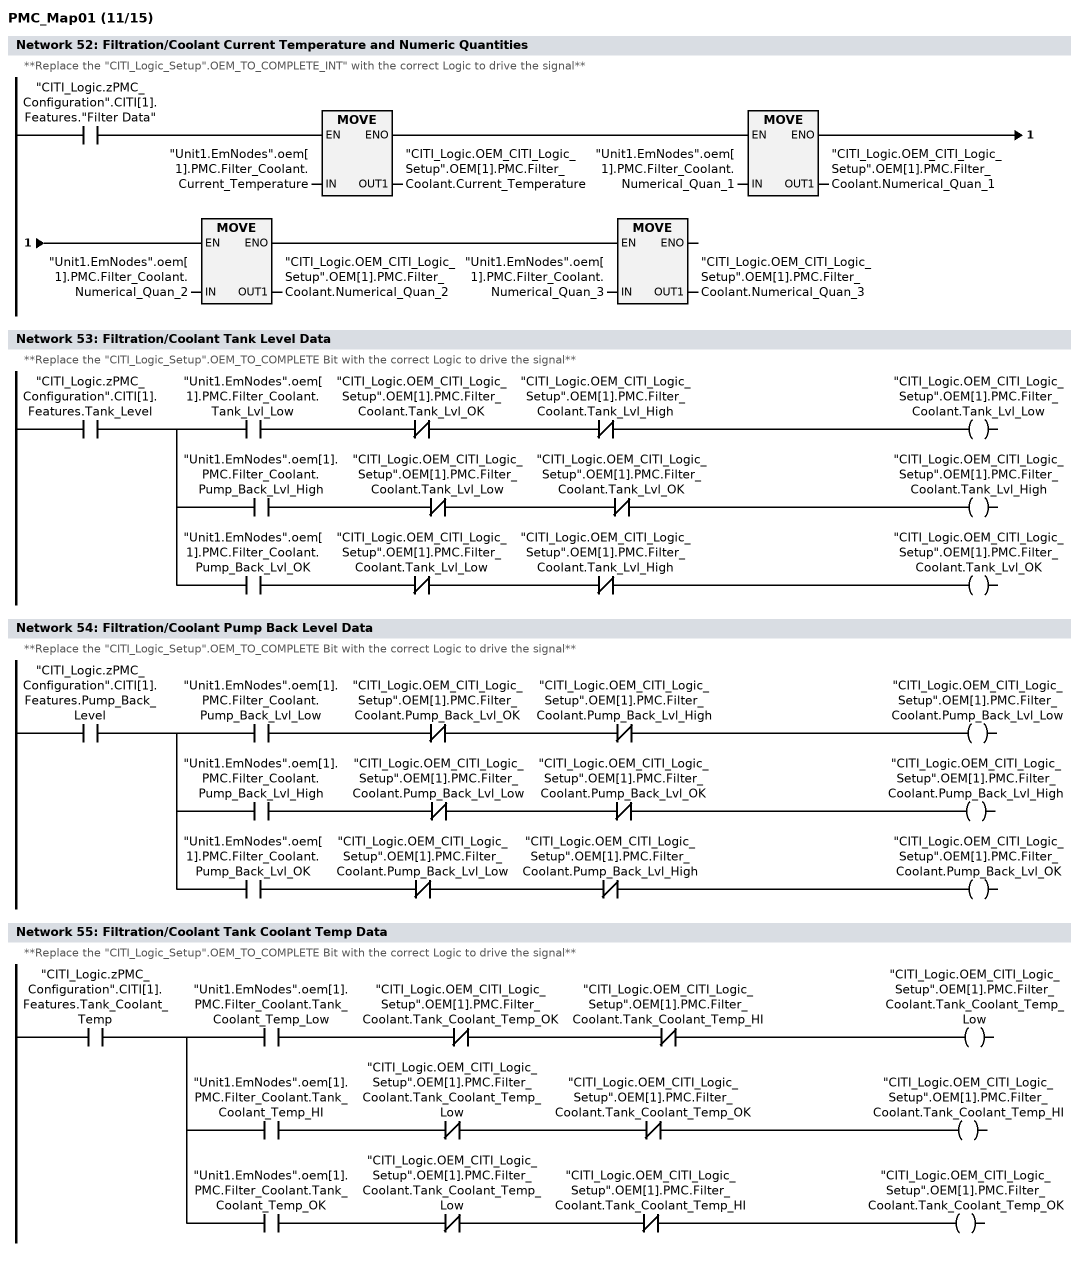
   RUNG wire#powerrail
      Contact( "CITI_Logic.zPMC_Configuration".CITI[1].Features."Filter Data" )
      Move(in := "Unit1.EmNodes".oem[1].PMC.Filter_Coolant.Current_Temperature, out1 => "CITI_Logic.OEM_CITI_Logic_Setup".OEM[1].PMC.Filter_Coolant.Current_Temperature)
      Move(in := "Unit1.EmNodes".oem[1].PMC.Filter_Coolant.Numerical_Quan_1, out1 => "CITI_Logic.OEM_CITI_Logic_Setup".OEM[1].PMC.Filter_Coolant.Numerical_Quan_1)
      Move(in := "Unit1.EmNodes".oem[1].PMC.Filter_Coolant.Numerical_Quan_2, out1 => "CITI_Logic.OEM_CITI_Logic_Setup".OEM[1].PMC.Filter_Coolant.Numerical_Quan_2)
      Move(in := "Unit1.EmNodes".oem[1].PMC.Filter_Coolant.Numerical_Quan_3, out1 => "CITI_Logic.OEM_CITI_Logic_Setup".OEM[1].PMC.Filter_Coolant.Numerical_Quan_3)
   END_RUNG
   // the same network as SCL:
   IF "CITI_Logic.zPMC_Configuration".CITI[1].Features."Filter Data" THEN
       "CITI_Logic.OEM_CITI_Logic_Setup".OEM[1].PMC.Filter_Coolant.Current_Temperature := "Unit1.EmNodes".oem[1].PMC.Filter_Coolant.Current_Temperature;
       "CITI_Logic.OEM_CITI_Logic_Setup".OEM[1].PMC.Filter_Coolant.Numerical_Quan_1 := "Unit1.EmNodes".oem[1].PMC.Filter_Coolant.Numerical_Quan_1;
       "CITI_Logic.OEM_CITI_Logic_Setup".OEM[1].PMC.Filter_Coolant.Numerical_Quan_2 := "Unit1.EmNodes".oem[1].PMC.Filter_Coolant.Numerical_Quan_2;
       "CITI_Logic.OEM_CITI_Logic_Setup".OEM[1].PMC.Filter_Coolant.Numerical_Quan_3 := "Unit1.EmNodes".oem[1].PMC.Filter_Coolant.Numerical_Quan_3;
   END_IF;
END_REGION

REGION Network 53: Filtration/Coolant Tank Level Data
   // **Replace the "CITI_Logic_Setup".OEM_TO_COMPLETE Bit with the correct Logic to drive the signal**
   RUNG wire#powerrail
      Contact( "CITI_Logic.zPMC_Configuration".CITI[1].Features.Tank_Level )
      wire#w1
      Contact( "Unit1.EmNodes".oem[1].PMC.Filter_Coolant.Tank_Lvl_Low )
      I_Contact( "CITI_Logic.OEM_CITI_Logic_Setup".OEM[1].PMC.Filter_Coolant.Tank_Lvl_OK )
      I_Contact( "CITI_Logic.OEM_CITI_Logic_Setup".OEM[1].PMC.Filter_Coolant.Tank_Lvl_High )
      Coil( "CITI_Logic.OEM_CITI_Logic_Setup".OEM[1].PMC.Filter_Coolant.Tank_Lvl_Low )
   END_RUNG
   RUNG wire#w1
      Contact( "Unit1.EmNodes".oem[1].PMC.Filter_Coolant.Pump_Back_Lvl_High )
      I_Contact( "CITI_Logic.OEM_CITI_Logic_Setup".OEM[1].PMC.Filter_Coolant.Tank_Lvl_Low )
      I_Contact( "CITI_Logic.OEM_CITI_Logic_Setup".OEM[1].PMC.Filter_Coolant.Tank_Lvl_OK )
      Coil( "CITI_Logic.OEM_CITI_Logic_Setup".OEM[1].PMC.Filter_Coolant.Tank_Lvl_High )
   END_RUNG
   RUNG wire#w1
      Contact( "Unit1.EmNodes".oem[1].PMC.Filter_Coolant.Pump_Back_Lvl_OK )
      I_Contact( "CITI_Logic.OEM_CITI_Logic_Setup".OEM[1].PMC.Filter_Coolant.Tank_Lvl_Low )
      I_Contact( "CITI_Logic.OEM_CITI_Logic_Setup".OEM[1].PMC.Filter_Coolant.Tank_Lvl_High )
      Coil( "CITI_Logic.OEM_CITI_Logic_Setup".OEM[1].PMC.Filter_Coolant.Tank_Lvl_OK )
   END_RUNG
   // the same network as SCL:
   "CITI_Logic.OEM_CITI_Logic_Setup".OEM[1].PMC.Filter_Coolant.Tank_Lvl_Low := "CITI_Logic.zPMC_Configuration".CITI[1].Features.Tank_Level AND "Unit1.EmNodes".oem[1].PMC.Filter_Coolant.Tank_Lvl_Low AND NOT "CITI_Logic.OEM_CITI_Logic_Setup".OEM[1].PMC.Filter_Coolant.Tank_Lvl_OK AND NOT "CITI_Logic.OEM_CITI_Logic_Setup".OEM[1].PMC.Filter_Coolant.Tank_Lvl_High;
   "CITI_Logic.OEM_CITI_Logic_Setup".OEM[1].PMC.Filter_Coolant.Tank_Lvl_High := "CITI_Logic.zPMC_Configuration".CITI[1].Features.Tank_Level AND "Unit1.EmNodes".oem[1].PMC.Filter_Coolant.Pump_Back_Lvl_High AND NOT "CITI_Logic.OEM_CITI_Logic_Setup".OEM[1].PMC.Filter_Coolant.Tank_Lvl_Low AND NOT "CITI_Logic.OEM_CITI_Logic_Setup".OEM[1].PMC.Filter_Coolant.Tank_Lvl_OK;
   "CITI_Logic.OEM_CITI_Logic_Setup".OEM[1].PMC.Filter_Coolant.Tank_Lvl_OK := "CITI_Logic.zPMC_Configuration".CITI[1].Features.Tank_Level AND "Unit1.EmNodes".oem[1].PMC.Filter_Coolant.Pump_Back_Lvl_OK AND NOT "CITI_Logic.OEM_CITI_Logic_Setup".OEM[1].PMC.Filter_Coolant.Tank_Lvl_Low AND NOT "CITI_Logic.OEM_CITI_Logic_Setup".OEM[1].PMC.Filter_Coolant.Tank_Lvl_High;
END_REGION

REGION Network 54: Filtration/Coolant Pump Back Level Data
   // **Replace the "CITI_Logic_Setup".OEM_TO_COMPLETE Bit with the correct Logic to drive the signal**
   RUNG wire#powerrail
      Contact( "CITI_Logic.zPMC_Configuration".CITI[1].Features.Pump_Back_Level )
      wire#w1
      Contact( "Unit1.EmNodes".oem[1].PMC.Filter_Coolant.Pump_Back_Lvl_Low )
      I_Contact( "CITI_Logic.OEM_CITI_Logic_Setup".OEM[1].PMC.Filter_Coolant.Pump_Back_Lvl_OK )
      I_Contact( "CITI_Logic.OEM_CITI_Logic_Setup".OEM[1].PMC.Filter_Coolant.Pump_Back_Lvl_High )
      Coil( "CITI_Logic.OEM_CITI_Logic_Setup".OEM[1].PMC.Filter_Coolant.Pump_Back_Lvl_Low )
   END_RUNG
   RUNG wire#w1
      Contact( "Unit1.EmNodes".oem[1].PMC.Filter_Coolant.Pump_Back_Lvl_High )
      I_Contact( "CITI_Logic.OEM_CITI_Logic_Setup".OEM[1].PMC.Filter_Coolant.Pump_Back_Lvl_Low )
      I_Contact( "CITI_Logic.OEM_CITI_Logic_Setup".OEM[1].PMC.Filter_Coolant.Pump_Back_Lvl_OK )
      Coil( "CITI_Logic.OEM_CITI_Logic_Setup".OEM[1].PMC.Filter_Coolant.Pump_Back_Lvl_High )
   END_RUNG
   RUNG wire#w1
      Contact( "Unit1.EmNodes".oem[1].PMC.Filter_Coolant.Pump_Back_Lvl_OK )
      I_Contact( "CITI_Logic.OEM_CITI_Logic_Setup".OEM[1].PMC.Filter_Coolant.Pump_Back_Lvl_Low )
      I_Contact( "CITI_Logic.OEM_CITI_Logic_Setup".OEM[1].PMC.Filter_Coolant.Pump_Back_Lvl_High )
      Coil( "CITI_Logic.OEM_CITI_Logic_Setup".OEM[1].PMC.Filter_Coolant.Pump_Back_Lvl_OK )
   END_RUNG
   // the same network as SCL:
   "CITI_Logic.OEM_CITI_Logic_Setup".OEM[1].PMC.Filter_Coolant.Pump_Back_Lvl_Low := "CITI_Logic.zPMC_Configuration".CITI[1].Features.Pump_Back_Level AND "Unit1.EmNodes".oem[1].PMC.Filter_Coolant.Pump_Back_Lvl_Low AND NOT "CITI_Logic.OEM_CITI_Logic_Setup".OEM[1].PMC.Filter_Coolant.Pump_Back_Lvl_OK AND NOT "CITI_Logic.OEM_CITI_Logic_Setup".OEM[1].PMC.Filter_Coolant.Pump_Back_Lvl_High;
   "CITI_Logic.OEM_CITI_Logic_Setup".OEM[1].PMC.Filter_Coolant.Pump_Back_Lvl_High := "CITI_Logic.zPMC_Configuration".CITI[1].Features.Pump_Back_Level AND "Unit1.EmNodes".oem[1].PMC.Filter_Coolant.Pump_Back_Lvl_High AND NOT "CITI_Logic.OEM_CITI_Logic_Setup".OEM[1].PMC.Filter_Coolant.Pump_Back_Lvl_Low AND NOT "CITI_Logic.OEM_CITI_Logic_Setup".OEM[1].PMC.Filter_Coolant.Pump_Back_Lvl_OK;
   "CITI_Logic.OEM_CITI_Logic_Setup".OEM[1].PMC.Filter_Coolant.Pump_Back_Lvl_OK := "CITI_Logic.zPMC_Configuration".CITI[1].Features.Pump_Back_Level AND "Unit1.EmNodes".oem[1].PMC.Filter_Coolant.Pump_Back_Lvl_OK AND NOT "CITI_Logic.OEM_CITI_Logic_Setup".OEM[1].PMC.Filter_Coolant.Pump_Back_Lvl_Low AND NOT "CITI_Logic.OEM_CITI_Logic_Setup".OEM[1].PMC.Filter_Coolant.Pump_Back_Lvl_High;
END_REGION

REGION Network 55: Filtration/Coolant Tank Coolant Temp Data
   // **Replace the "CITI_Logic_Setup".OEM_TO_COMPLETE Bit with the correct Logic to drive the signal**
   RUNG wire#powerrail
      Contact( "CITI_Logic.zPMC_Configuration".CITI[1].Features.Tank_Coolant_Temp )
      wire#w1
      Contact( "Unit1.EmNodes".oem[1].PMC.Filter_Coolant.Tank_Coolant_Temp_Low )
      I_Contact( "CITI_Logic.OEM_CITI_Logic_Setup".OEM[1].PMC.Filter_Coolant.Tank_Coolant_Temp_OK )
      I_Contact( "CITI_Logic.OEM_CITI_Logic_Setup".OEM[1].PMC.Filter_Coolant.Tank_Coolant_Temp_HI )
      Coil( "CITI_Logic.OEM_CITI_Logic_Setup".OEM[1].PMC.Filter_Coolant.Tank_Coolant_Temp_Low )
   END_RUNG
   RUNG wire#w1
      Contact( "Unit1.EmNodes".oem[1].PMC.Filter_Coolant.Tank_Coolant_Temp_HI )
      I_Contact( "CITI_Logic.OEM_CITI_Logic_Setup".OEM[1].PMC.Filter_Coolant.Tank_Coolant_Temp_Low )
      I_Contact( "CITI_Logic.OEM_CITI_Logic_Setup".OEM[1].PMC.Filter_Coolant.Tank_Coolant_Temp_OK )
      Coil( "CITI_Logic.OEM_CITI_Logic_Setup".OEM[1].PMC.Filter_Coolant.Tank_Coolant_Temp_HI )
   END_RUNG
   RUNG wire#w1
      Contact( "Unit1.EmNodes".oem[1].PMC.Filter_Coolant.Tank_Coolant_Temp_OK )
      I_Contact( "CITI_Logic.OEM_CITI_Logic_Setup".OEM[1].PMC.Filter_Coolant.Tank_Coolant_Temp_Low )
      I_Contact( "CITI_Logic.OEM_CITI_Logic_Setup".OEM[1].PMC.Filter_Coolant.Tank_Coolant_Temp_HI )
      Coil( "CITI_Logic.OEM_CITI_Logic_Setup".OEM[1].PMC.Filter_Coolant.Tank_Coolant_Temp_OK )
   END_RUNG
   // the same network as SCL:
   "CITI_Logic.OEM_CITI_Logic_Setup".OEM[1].PMC.Filter_Coolant.Tank_Coolant_Temp_Low := "CITI_Logic.zPMC_Configuration".CITI[1].Features.Tank_Coolant_Temp AND "Unit1.EmNodes".oem[1].PMC.Filter_Coolant.Tank_Coolant_Temp_Low AND NOT "CITI_Logic.OEM_CITI_Logic_Setup".OEM[1].PMC.Filter_Coolant.Tank_Coolant_Temp_OK AND NOT "CITI_Logic.OEM_CITI_Logic_Setup".OEM[1].PMC.Filter_Coolant.Tank_Coolant_Temp_HI;
   "CITI_Logic.OEM_CITI_Logic_Setup".OEM[1].PMC.Filter_Coolant.Tank_Coolant_Temp_HI := "CITI_Logic.zPMC_Configuration".CITI[1].Features.Tank_Coolant_Temp AND "Unit1.EmNodes".oem[1].PMC.Filter_Coolant.Tank_Coolant_Temp_HI AND NOT "CITI_Logic.OEM_CITI_Logic_Setup".OEM[1].PMC.Filter_Coolant.Tank_Coolant_Temp_Low AND NOT "CITI_Logic.OEM_CITI_Logic_Setup".OEM[1].PMC.Filter_Coolant.Tank_Coolant_Temp_OK;
   "CITI_Logic.OEM_CITI_Logic_Setup".OEM[1].PMC.Filter_Coolant.Tank_Coolant_Temp_OK := "CITI_Logic.zPMC_Configuration".CITI[1].Features.Tank_Coolant_Temp AND "Unit1.EmNodes".oem[1].PMC.Filter_Coolant.Tank_Coolant_Temp_OK AND NOT "CITI_Logic.OEM_CITI_Logic_Setup".OEM[1].PMC.Filter_Coolant.Tank_Coolant_Temp_Low AND NOT "CITI_Logic.OEM_CITI_Logic_Setup".OEM[1].PMC.Filter_Coolant.Tank_Coolant_Temp_HI;
END_REGION

REGION Network 56: CMM Specific Data
   // **Replace the "CITI_Logic_Setup".OEM_TO_COMPLETE Bit and "CITI_Logic_Setup".OEM_TO_COMPLETE_INT" with the correct Logic to drive the signal**
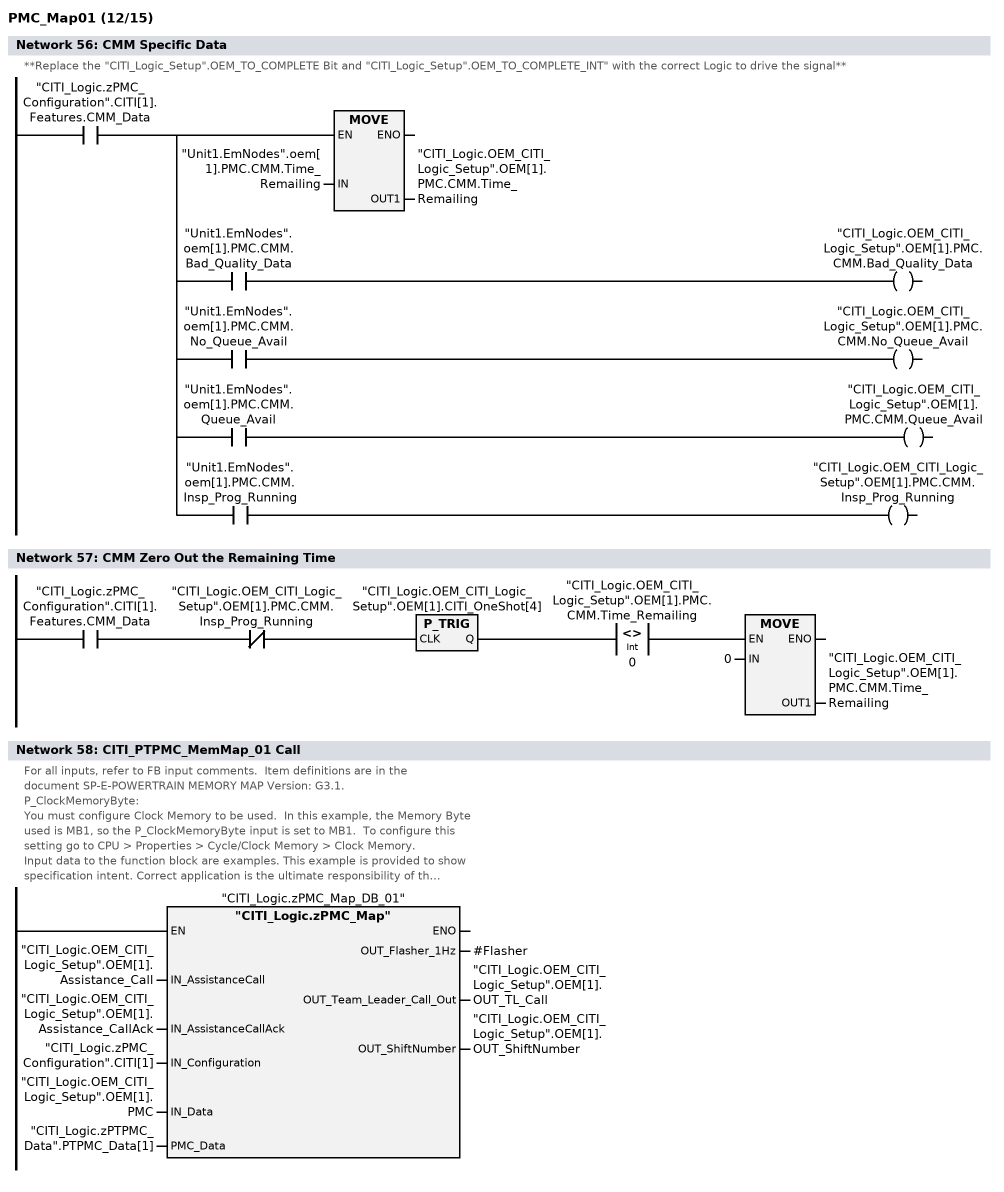
   RUNG wire#powerrail
      Contact( "CITI_Logic.zPMC_Configuration".CITI[1].Features.CMM_Data )
      wire#w1
      Move(in := "Unit1.EmNodes".oem[1].PMC.CMM.Time_Remailing, out1 => "CITI_Logic.OEM_CITI_Logic_Setup".OEM[1].PMC.CMM.Time_Remailing)
   END_RUNG
   RUNG wire#w1
      Contact( "Unit1.EmNodes".oem[1].PMC.CMM.Bad_Quality_Data )
      Coil( "CITI_Logic.OEM_CITI_Logic_Setup".OEM[1].PMC.CMM.Bad_Quality_Data )
   END_RUNG
   RUNG wire#w1
      Contact( "Unit1.EmNodes".oem[1].PMC.CMM.No_Queue_Avail )
      Coil( "CITI_Logic.OEM_CITI_Logic_Setup".OEM[1].PMC.CMM.No_Queue_Avail )
   END_RUNG
   RUNG wire#w1
      Contact( "Unit1.EmNodes".oem[1].PMC.CMM.Queue_Avail )
      Coil( "CITI_Logic.OEM_CITI_Logic_Setup".OEM[1].PMC.CMM.Queue_Avail )
   END_RUNG
   RUNG wire#w1
      Contact( "Unit1.EmNodes".oem[1].PMC.CMM.Insp_Prog_Running )
      Coil( "CITI_Logic.OEM_CITI_Logic_Setup".OEM[1].PMC.CMM.Insp_Prog_Running )
   END_RUNG
   // the same network as SCL:
   IF "CITI_Logic.zPMC_Configuration".CITI[1].Features.CMM_Data THEN
       "CITI_Logic.OEM_CITI_Logic_Setup".OEM[1].PMC.CMM.Time_Remailing := "Unit1.EmNodes".oem[1].PMC.CMM.Time_Remailing;
   END_IF;
   "CITI_Logic.OEM_CITI_Logic_Setup".OEM[1].PMC.CMM.Bad_Quality_Data := "CITI_Logic.zPMC_Configuration".CITI[1].Features.CMM_Data AND "Unit1.EmNodes".oem[1].PMC.CMM.Bad_Quality_Data;
   "CITI_Logic.OEM_CITI_Logic_Setup".OEM[1].PMC.CMM.No_Queue_Avail := "CITI_Logic.zPMC_Configuration".CITI[1].Features.CMM_Data AND "Unit1.EmNodes".oem[1].PMC.CMM.No_Queue_Avail;
   "CITI_Logic.OEM_CITI_Logic_Setup".OEM[1].PMC.CMM.Queue_Avail := "CITI_Logic.zPMC_Configuration".CITI[1].Features.CMM_Data AND "Unit1.EmNodes".oem[1].PMC.CMM.Queue_Avail;
   "CITI_Logic.OEM_CITI_Logic_Setup".OEM[1].PMC.CMM.Insp_Prog_Running := "CITI_Logic.zPMC_Configuration".CITI[1].Features.CMM_Data AND "Unit1.EmNodes".oem[1].PMC.CMM.Insp_Prog_Running;
END_REGION

REGION Network 57: CMM Zero Out the Remaining Time
   RUNG wire#powerrail
      Contact( "CITI_Logic.zPMC_Configuration".CITI[1].Features.CMM_Data )
      I_Contact( "CITI_Logic.OEM_CITI_Logic_Setup".OEM[1].PMC.CMM.Insp_Prog_Running )
      P_Trig( "CITI_Logic.OEM_CITI_Logic_Setup".OEM[1].CITI_OneShot[4] )
      { S7_Templates := "SrcType := Int" } NE_Contact(in1 := "CITI_Logic.OEM_CITI_Logic_Setup".OEM[1].PMC.CMM.Time_Remailing, in2 := 0)
      { S7_GenerateENO := "TRUE" } Move(in := 0, out1 => "CITI_Logic.OEM_CITI_Logic_Setup".OEM[1].PMC.CMM.Time_Remailing)
   END_RUNG
   // the same network as SCL:
   #_w1 := "CITI_Logic.zPMC_Configuration".CITI[1].Features.CMM_Data AND NOT "CITI_Logic.OEM_CITI_Logic_Setup".OEM[1].PMC.CMM.Insp_Prog_Running;
   #_w2 := #_w1 AND NOT "CITI_Logic.OEM_CITI_Logic_Setup".OEM[1].CITI_OneShot[4];   // rising edge
   "CITI_Logic.OEM_CITI_Logic_Setup".OEM[1].CITI_OneShot[4] := #_w1;
   IF #_w2 AND ("CITI_Logic.OEM_CITI_Logic_Setup".OEM[1].PMC.CMM.Time_Remailing <> 0) THEN
       "CITI_Logic.OEM_CITI_Logic_Setup".OEM[1].PMC.CMM.Time_Remailing := 0;
   END_IF;
END_REGION

REGION Network 58: CITI_PTPMC_MemMap_01 Call
   // For all inputs, refer to FB input comments.  Item definitions are in the 
   // document SP-E-POWERTRAIN MEMORY MAP Version: G3.1.
   // 
   // P_ClockMemoryByte:
   // You must configure Clock Memory to be used.  In this example, the Memory Byte 
   // used is MB1, so the P_ClockMemoryByte input is set to MB1.  To configure this 
   // setting go to CPU > Properties > Cycle/Clock Memory > Clock Memory.
   // 
   // Input data to the function block are examples. This example is provided to show 
   // specification intent. Correct application is the ultimate responsibility of the 
   // OEM. 
   // 
   // See the accompanying documentation for more information. For questions, please 
   // contact the GMPT Controls/I.T. Integration Engineer for your project.
   RUNG wire#powerrail
      "CITI_Logic.zPMC_Map_DB_01"(IN_AssistanceCall := "CITI_Logic.OEM_CITI_Logic_Setup".OEM[1].Assistance_Call, IN_AssistanceCallAck := "CITI_Logic.OEM_CITI_Logic_Setup".OEM[1].Assistance_CallAck, IN_Configuration := "CITI_Logic.zPMC_Configuration".CITI[1], IN_Data := "CITI_Logic.OEM_CITI_Logic_Setup".OEM[1].PMC, PMC_Data := "CITI_Logic.zPTPMC_Data".PTPMC_Data[1], OUT_Flasher_1Hz => #Flasher, OUT_Team_Leader_Call_Out => "CITI_Logic.OEM_CITI_Logic_Setup".OEM[1].OUT_TL_Call, OUT_ShiftNumber => "CITI_Logic.OEM_CITI_Logic_Setup".OEM[1].OUT_ShiftNumber)
   END_RUNG
   // the same network as SCL:
   "CITI_Logic.zPMC_Map_DB_01"(IN_AssistanceCall := "CITI_Logic.OEM_CITI_Logic_Setup".OEM[1].Assistance_Call,   // "CITI_Logic.zPMC_Map"
                           IN_AssistanceCallAck := "CITI_Logic.OEM_CITI_Logic_Setup".OEM[1].Assistance_CallAck,
                           IN_Configuration := "CITI_Logic.zPMC_Configuration".CITI[1],
                           IN_Data := "CITI_Logic.OEM_CITI_Logic_Setup".OEM[1].PMC,
                           PMC_Data := "CITI_Logic.zPTPMC_Data".PTPMC_Data[1],
                           OUT_Flasher_1Hz => #Flasher,
                           OUT_Team_Leader_Call_Out => "CITI_Logic.OEM_CITI_Logic_Setup".OEM[1].OUT_TL_Call,
                           OUT_ShiftNumber => "CITI_Logic.OEM_CITI_Logic_Setup".OEM[1].OUT_ShiftNumber);
END_REGION

REGION Network 59: Stack Light: Red Light
   // All stacklights should be driven by bits in the Memory Map.  The following is 
   // an example, however, your particular implementation must follow the rules 
   // determined by the particular project or common approach.  This will be dictated 
   // by the GMPT controls engineer.  The logic below is an EXAMPLE ONLY.
   // 
   // Red light consists of flashing and solid commands, where flashing is 
   // prioritized, and then summarized in the output.
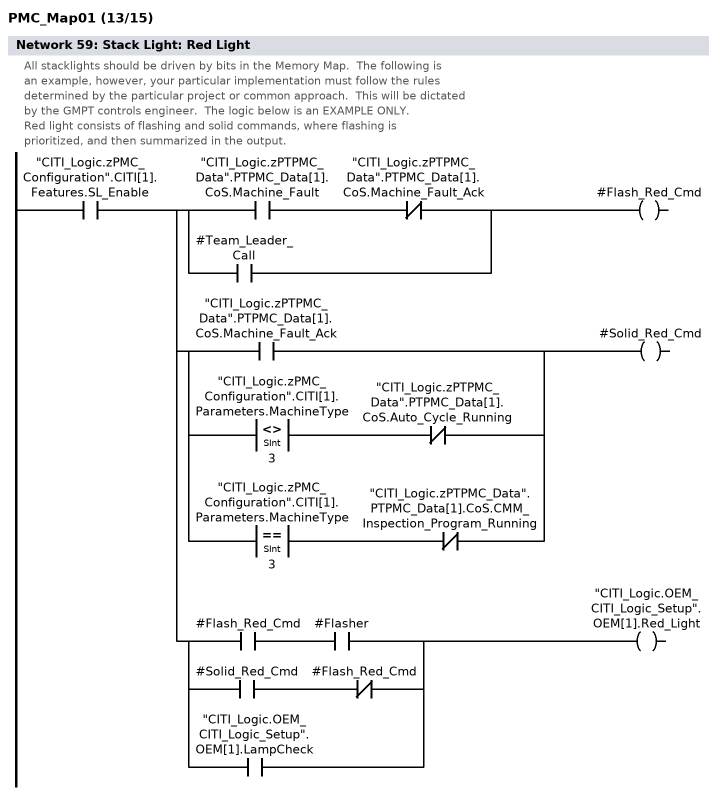
   RUNG wire#powerrail
      Contact( "CITI_Logic.zPMC_Configuration".CITI[1].Features.SL_Enable )
      wire#w1
      Contact( "CITI_Logic.zPTPMC_Data".PTPMC_Data[1].CoS.Machine_Fault )
      I_Contact( "CITI_Logic.zPTPMC_Data".PTPMC_Data[1].CoS.Machine_Fault_Ack )
      wire#w2
      Coil( #Flash_Red_Cmd )
   END_RUNG
   RUNG wire#w1
      Contact( #Team_Leader_Call )
   END_RUNG wire#w2
   RUNG wire#w1
      Contact( "CITI_Logic.zPTPMC_Data".PTPMC_Data[1].CoS.Machine_Fault_Ack )
      wire#w3
      Coil( #Solid_Red_Cmd )
   END_RUNG
   RUNG wire#w1
      { S7_Templates := "SrcType := SInt" } NE_Contact(in1 := "CITI_Logic.zPMC_Configuration".CITI[1].Parameters.MachineType, in2 := 3)
      I_Contact( "CITI_Logic.zPTPMC_Data".PTPMC_Data[1].CoS.Auto_Cycle_Running )
   END_RUNG wire#w3
   RUNG wire#w1
      { S7_Templates := "SrcType := SInt" } EQ_Contact(in1 := "CITI_Logic.zPMC_Configuration".CITI[1].Parameters.MachineType, in2 := 3)
      I_Contact( "CITI_Logic.zPTPMC_Data".PTPMC_Data[1].CoS.CMM_Inspection_Program_Running )
   END_RUNG wire#w3
   RUNG wire#w1
      Contact( #Flash_Red_Cmd )
      Contact( #Flasher )
      wire#w4
      Coil( "CITI_Logic.OEM_CITI_Logic_Setup".OEM[1].Red_Light )
   END_RUNG
   RUNG wire#w1
      Contact( #Solid_Red_Cmd )
      I_Contact( #Flash_Red_Cmd )
   END_RUNG wire#w4
   RUNG wire#w1
      Contact( "CITI_Logic.OEM_CITI_Logic_Setup".OEM[1].LampCheck )
   END_RUNG wire#w4
   // the same network as SCL:
   #Flash_Red_Cmd := "CITI_Logic.zPMC_Configuration".CITI[1].Features.SL_Enable AND (("CITI_Logic.zPTPMC_Data".PTPMC_Data[1].CoS.Machine_Fault AND NOT "CITI_Logic.zPTPMC_Data".PTPMC_Data[1].CoS.Machine_Fault_Ack) OR #Team_Leader_Call);
   #Solid_Red_Cmd := "CITI_Logic.zPMC_Configuration".CITI[1].Features.SL_Enable AND ("CITI_Logic.zPTPMC_Data".PTPMC_Data[1].CoS.Machine_Fault_Ack OR (("CITI_Logic.zPMC_Configuration".CITI[1].Parameters.MachineType <> 3) AND NOT "CITI_Logic.zPTPMC_Data".PTPMC_Data[1].CoS.Auto_Cycle_Running) OR (("CITI_Logic.zPMC_Configuration".CITI[1].Parameters.MachineType = 3) AND NOT "CITI_Logic.zPTPMC_Data".PTPMC_Data[1].CoS.CMM_Inspection_Program_Running));
   "CITI_Logic.OEM_CITI_Logic_Setup".OEM[1].Red_Light := "CITI_Logic.zPMC_Configuration".CITI[1].Features.SL_Enable AND ((#Flash_Red_Cmd AND #Flasher) OR (#Solid_Red_Cmd AND NOT #Flash_Red_Cmd) OR "CITI_Logic.OEM_CITI_Logic_Setup".OEM[1].LampCheck);
END_REGION

REGION Network 60: Stack Light: Yellow Light
   // All stacklights should be driven by bits in the Memory Map.  The following is 
   // an example, however, your particular implementation must follow the rules 
   // determined by the particular project or common approach.  This will be dictated 
   // by the GMPT controls engineer.  The logic below is an EXAMPLE ONLY.
   // 
   // Yellow light consists of flashing and solid commands, where flashing is 
   // prioritized, and then summarized in the output.
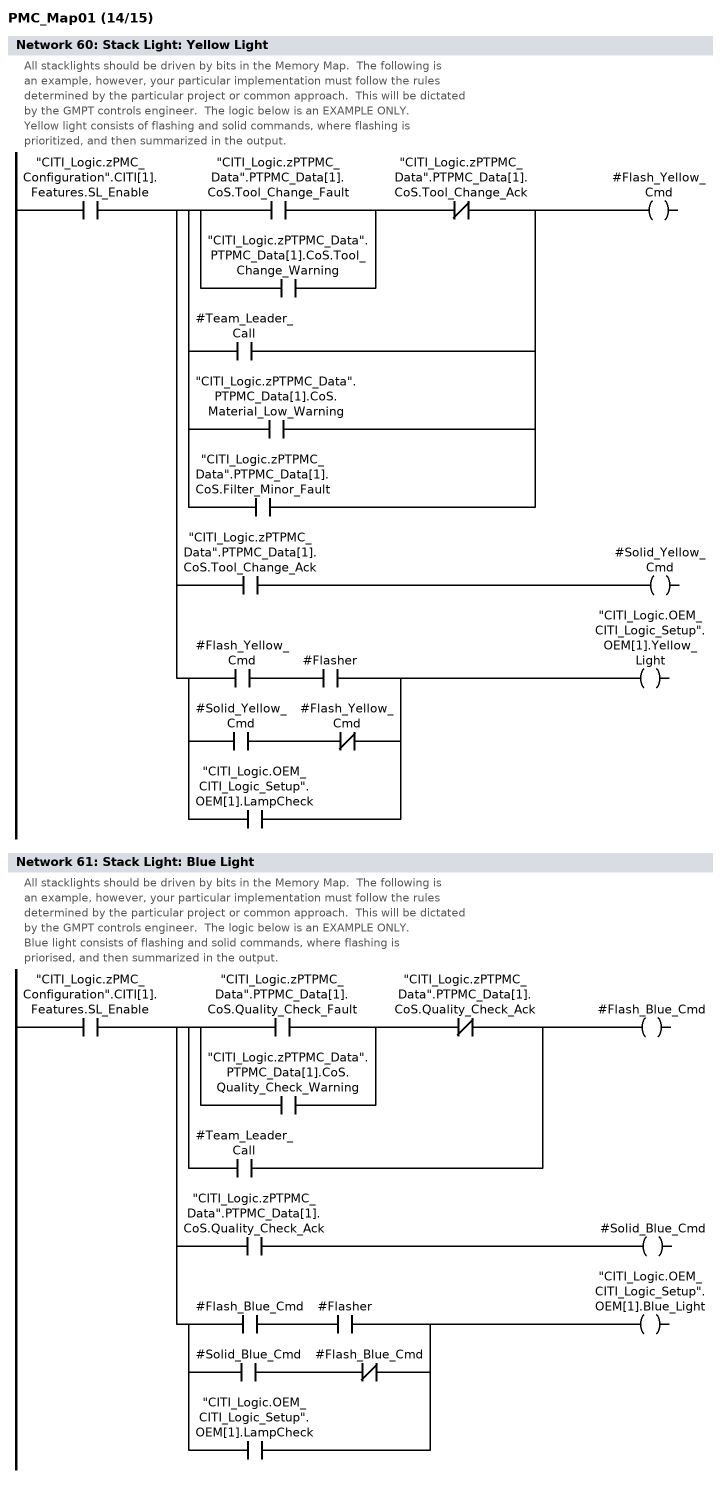
   RUNG wire#powerrail
      Contact( "CITI_Logic.zPMC_Configuration".CITI[1].Features.SL_Enable )
      wire#w1
      Contact( "CITI_Logic.zPTPMC_Data".PTPMC_Data[1].CoS.Tool_Change_Fault )
      wire#w2
      I_Contact( "CITI_Logic.zPTPMC_Data".PTPMC_Data[1].CoS.Tool_Change_Ack )
      wire#w3
      Coil( #Flash_Yellow_Cmd )
   END_RUNG
   RUNG wire#w1
      Contact( "CITI_Logic.zPTPMC_Data".PTPMC_Data[1].CoS.Tool_Change_Warning )
   END_RUNG wire#w2
   RUNG wire#w1
      Contact( #Team_Leader_Call )
   END_RUNG wire#w3
   RUNG wire#w1
      Contact( "CITI_Logic.zPTPMC_Data".PTPMC_Data[1].CoS.Material_Low_Warning )
   END_RUNG wire#w3
   RUNG wire#w1
      Contact( "CITI_Logic.zPTPMC_Data".PTPMC_Data[1].CoS.Filter_Minor_Fault )
   END_RUNG wire#w3
   RUNG wire#w1
      Contact( "CITI_Logic.zPTPMC_Data".PTPMC_Data[1].CoS.Tool_Change_Ack )
      Coil( #Solid_Yellow_Cmd )
   END_RUNG
   RUNG wire#w1
      Contact( #Flash_Yellow_Cmd )
      Contact( #Flasher )
      wire#w4
      Coil( "CITI_Logic.OEM_CITI_Logic_Setup".OEM[1].Yellow_Light )
   END_RUNG
   RUNG wire#w1
      Contact( #Solid_Yellow_Cmd )
      I_Contact( #Flash_Yellow_Cmd )
   END_RUNG wire#w4
   RUNG wire#w1
      Contact( "CITI_Logic.OEM_CITI_Logic_Setup".OEM[1].LampCheck )
   END_RUNG wire#w4
   // the same network as SCL:
   #Flash_Yellow_Cmd := "CITI_Logic.zPMC_Configuration".CITI[1].Features.SL_Enable AND ((("CITI_Logic.zPTPMC_Data".PTPMC_Data[1].CoS.Tool_Change_Fault OR "CITI_Logic.zPTPMC_Data".PTPMC_Data[1].CoS.Tool_Change_Warning) AND NOT "CITI_Logic.zPTPMC_Data".PTPMC_Data[1].CoS.Tool_Change_Ack) OR #Team_Leader_Call OR "CITI_Logic.zPTPMC_Data".PTPMC_Data[1].CoS.Material_Low_Warning OR "CITI_Logic.zPTPMC_Data".PTPMC_Data[1].CoS.Filter_Minor_Fault);
   #Solid_Yellow_Cmd := "CITI_Logic.zPMC_Configuration".CITI[1].Features.SL_Enable AND "CITI_Logic.zPTPMC_Data".PTPMC_Data[1].CoS.Tool_Change_Ack;
   "CITI_Logic.OEM_CITI_Logic_Setup".OEM[1].Yellow_Light := "CITI_Logic.zPMC_Configuration".CITI[1].Features.SL_Enable AND ((#Flash_Yellow_Cmd AND #Flasher) OR (#Solid_Yellow_Cmd AND NOT #Flash_Yellow_Cmd) OR "CITI_Logic.OEM_CITI_Logic_Setup".OEM[1].LampCheck);
END_REGION

REGION Network 61: Stack Light: Blue Light
   // All stacklights should be driven by bits in the Memory Map.  The following is 
   // an example, however, your particular implementation must follow the rules 
   // determined by the particular project or common approach.  This will be dictated 
   // by the GMPT controls engineer.  The logic below is an EXAMPLE ONLY.
   // 
   // Blue light consists of flashing and solid commands, where flashing is 
   // priorised, and then summarized in the output.
   RUNG wire#powerrail
      Contact( "CITI_Logic.zPMC_Configuration".CITI[1].Features.SL_Enable )
      wire#w1
      Contact( "CITI_Logic.zPTPMC_Data".PTPMC_Data[1].CoS.Quality_Check_Fault )
      wire#w2
      I_Contact( "CITI_Logic.zPTPMC_Data".PTPMC_Data[1].CoS.Quality_Check_Ack )
      wire#w3
      Coil( #Flash_Blue_Cmd )
   END_RUNG
   RUNG wire#w1
      Contact( "CITI_Logic.zPTPMC_Data".PTPMC_Data[1].CoS.Quality_Check_Warning )
   END_RUNG wire#w2
   RUNG wire#w1
      Contact( #Team_Leader_Call )
   END_RUNG wire#w3
   RUNG wire#w1
      Contact( "CITI_Logic.zPTPMC_Data".PTPMC_Data[1].CoS.Quality_Check_Ack )
      Coil( #Solid_Blue_Cmd )
   END_RUNG
   RUNG wire#w1
      Contact( #Flash_Blue_Cmd )
      Contact( #Flasher )
      wire#w4
      Coil( "CITI_Logic.OEM_CITI_Logic_Setup".OEM[1].Blue_Light )
   END_RUNG
   RUNG wire#w1
      Contact( #Solid_Blue_Cmd )
      I_Contact( #Flash_Blue_Cmd )
   END_RUNG wire#w4
   RUNG wire#w1
      Contact( "CITI_Logic.OEM_CITI_Logic_Setup".OEM[1].LampCheck )
   END_RUNG wire#w4
   // the same network as SCL:
   #Flash_Blue_Cmd := "CITI_Logic.zPMC_Configuration".CITI[1].Features.SL_Enable AND ((("CITI_Logic.zPTPMC_Data".PTPMC_Data[1].CoS.Quality_Check_Fault OR "CITI_Logic.zPTPMC_Data".PTPMC_Data[1].CoS.Quality_Check_Warning) AND NOT "CITI_Logic.zPTPMC_Data".PTPMC_Data[1].CoS.Quality_Check_Ack) OR #Team_Leader_Call);
   #Solid_Blue_Cmd := "CITI_Logic.zPMC_Configuration".CITI[1].Features.SL_Enable AND "CITI_Logic.zPTPMC_Data".PTPMC_Data[1].CoS.Quality_Check_Ack;
   "CITI_Logic.OEM_CITI_Logic_Setup".OEM[1].Blue_Light := "CITI_Logic.zPMC_Configuration".CITI[1].Features.SL_Enable AND ((#Flash_Blue_Cmd AND #Flasher) OR (#Solid_Blue_Cmd AND NOT #Flash_Blue_Cmd) OR "CITI_Logic.OEM_CITI_Logic_Setup".OEM[1].LampCheck);
END_REGION

REGION Network 62: Stack Light: Green Light
   // All stacklights should be driven by bits in the Memory Map.  The following is 
   // an example, however, your particular implementation must follow the rules 
   // determined by the particular project or common approach.  This will be dictated 
   // by the GMPT controls engineer.  The logic below is an EXAMPLE ONLY.
   // 
   // Green light consists of flashing and solid commands, where flashing is 
   // prioritized, and then summarized in the output.
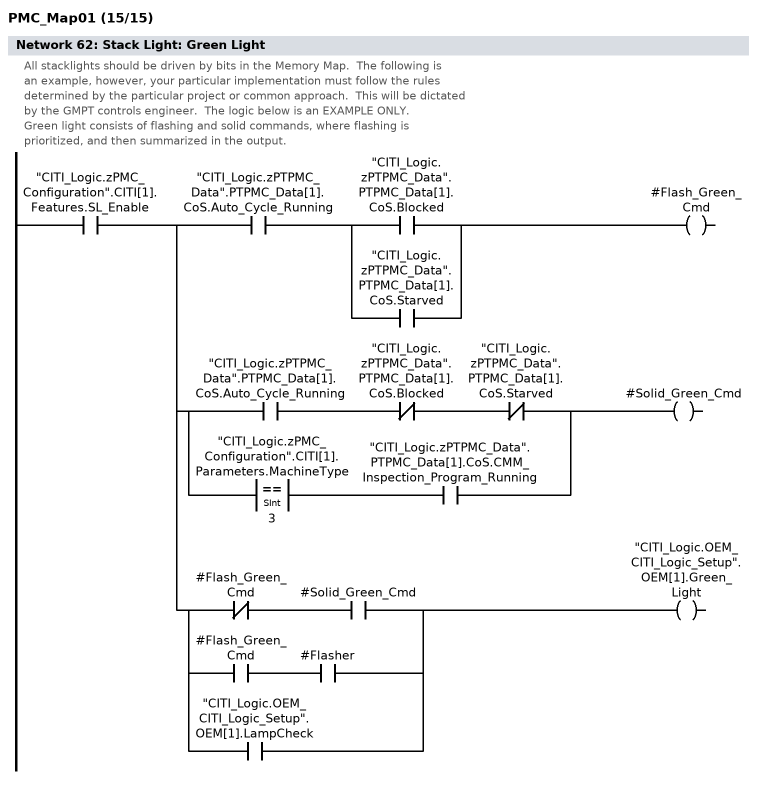
   RUNG wire#powerrail
      Contact( "CITI_Logic.zPMC_Configuration".CITI[1].Features.SL_Enable )
      wire#w1
      Contact( "CITI_Logic.zPTPMC_Data".PTPMC_Data[1].CoS.Auto_Cycle_Running )
      wire#w2
      Contact( "CITI_Logic.zPTPMC_Data".PTPMC_Data[1].CoS.Blocked )
      wire#w3
      Coil( #Flash_Green_Cmd )
   END_RUNG
   RUNG wire#w2
      Contact( "CITI_Logic.zPTPMC_Data".PTPMC_Data[1].CoS.Starved )
   END_RUNG wire#w3
   RUNG wire#w1
      Contact( "CITI_Logic.zPTPMC_Data".PTPMC_Data[1].CoS.Auto_Cycle_Running )
      I_Contact( "CITI_Logic.zPTPMC_Data".PTPMC_Data[1].CoS.Blocked )
      I_Contact( "CITI_Logic.zPTPMC_Data".PTPMC_Data[1].CoS.Starved )
      wire#w4
      Coil( #Solid_Green_Cmd )
   END_RUNG
   RUNG wire#w1
      { S7_Templates := "SrcType := SInt" } EQ_Contact(in1 := "CITI_Logic.zPMC_Configuration".CITI[1].Parameters.MachineType, in2 := 3)
      Contact( "CITI_Logic.zPTPMC_Data".PTPMC_Data[1].CoS.CMM_Inspection_Program_Running )
   END_RUNG wire#w4
   RUNG wire#w1
      I_Contact( #Flash_Green_Cmd )
      Contact( #Solid_Green_Cmd )
      wire#w5
      Coil( "CITI_Logic.OEM_CITI_Logic_Setup".OEM[1].Green_Light )
   END_RUNG
   RUNG wire#w1
      Contact( #Flash_Green_Cmd )
      Contact( #Flasher )
   END_RUNG wire#w5
   RUNG wire#w1
      Contact( "CITI_Logic.OEM_CITI_Logic_Setup".OEM[1].LampCheck )
   END_RUNG wire#w5
   // the same network as SCL:
   #Flash_Green_Cmd := "CITI_Logic.zPMC_Configuration".CITI[1].Features.SL_Enable AND "CITI_Logic.zPTPMC_Data".PTPMC_Data[1].CoS.Auto_Cycle_Running AND ("CITI_Logic.zPTPMC_Data".PTPMC_Data[1].CoS.Blocked OR "CITI_Logic.zPTPMC_Data".PTPMC_Data[1].CoS.Starved);
   #Solid_Green_Cmd := "CITI_Logic.zPMC_Configuration".CITI[1].Features.SL_Enable AND (("CITI_Logic.zPTPMC_Data".PTPMC_Data[1].CoS.Auto_Cycle_Running AND NOT "CITI_Logic.zPTPMC_Data".PTPMC_Data[1].CoS.Blocked AND NOT "CITI_Logic.zPTPMC_Data".PTPMC_Data[1].CoS.Starved) OR (("CITI_Logic.zPMC_Configuration".CITI[1].Parameters.MachineType = 3) AND "CITI_Logic.zPTPMC_Data".PTPMC_Data[1].CoS.CMM_Inspection_Program_Running));
   "CITI_Logic.OEM_CITI_Logic_Setup".OEM[1].Green_Light := "CITI_Logic.zPMC_Configuration".CITI[1].Features.SL_Enable AND ((NOT #Flash_Green_Cmd AND #Solid_Green_Cmd) OR (#Flash_Green_Cmd AND #Flasher) OR "CITI_Logic.OEM_CITI_Logic_Setup".OEM[1].LampCheck);
END_REGION
END_FUNCTION
